LIN {X 0,Y 189.496,Z 286.196,A -85,B 0,C 180,E1 -22198.72,E2 -22198.72} C_VEL
LIN {X 0,Y 187.932,Z 288.132,A -85,B 0,C 180,E1 -22200.913,E2 -22200.913} C_VEL
LIN {X 0,Y 186.648,Z 289.597,A -85,B 0,C 180,E1 -22203.139,E2 -22203.139} C_VEL
LIN {X 0,Y 185.608,Z 290.594,A -85,B 0,C 180,E1 -22205.386,E2 -22205.386} C_VEL
LIN {X 0,Y 184.681,Z 291.189,A -85,B 0,C 180,E1 -22207.633,E2 -22207.633} C_VEL
LIN {X 0,Y 183.977,Z 291.376,A -85,B 0,C 180,E1 -22209.892,E2 -22209.892} C_VEL
LIN {X 0,Y 183.377,Z 290.818,A -85,B 0,C 180,E1 -22213.366,E2 -22213.366} C_VEL
LIN {X 0,Y 183.176,Z 289.357,A -85,B 0,C 180,E1 -22216.692,E2 -22216.692} C_VEL
LIN {X 0,Y 183.239,Z 287.851,A -85,B 0,C 180,E1 -22218.945,E2 -22218.945} C_VEL
LIN {X 0,Y 183.723,Z 284.759,A -85,B 0,C 180,E1 -22222.307,E2 -22222.307} C_VEL
LIN {X 0,Y 184.434,Z 280.616,A -85,B 0,C 180,E1 -22225.63,E2 -22225.63} C_VEL
LIN {X 0,Y 185.666,Z 274.289,A -85,B 0,C 180,E1 -22229.459,E2 -22229.459} C_VEL
LIN {X 0,Y 187.209,Z 267.409,A -85,B 0,C 180,E1 -22232.69,E2 -22232.69} C_VEL
LIN {X 0,Y 188.876,Z 260.381,A -85,B 0,C 180,E1 -22235.338,E2 -22235.338} C_VEL
LIN {X 0,Y 190.904,Z 251.904,A -85,B 0,C 180,E1 -22237.936,E2 -22237.936} C_VEL
LIN {X 0,Y 193.116,Z 241.454,A -85,B 0,C 180,E1 -22240.485,E2 -22240.485} C_VEL
LIN {X 0,Y 195.098,Z 231.113,A -85,B 0,C 180,E1 -22242.483,E2 -22242.483} C_VEL
LIN {X 0,Y 196.96,Z 219.8,A -85,B 0,C 180,E1 -22244.201,E2 -22244.201} C_VEL
LIN {X 0,Y 198.45,Z 208.263,A -85,B 0,C 180,E1 -22245.535,E2 -22245.535} C_VEL
LIN {X 0,Y 199.783,Z 194.686,A -85,B 0,C 180,E1 -22246.631,E2 -22246.631} C_VEL
LIN {X 0,Y 200.565,Z 181.404,A -85,B 0,C 180,E1 -22247.294,E2 -22247.294} C_VEL
LIN {X 0,Y 202.876,Z 125.441,A -85,B 0,C 180,E1 -22249.181,E2 -22249.181} C_VEL
LIN {X 0,Y 196.139,Z 109.947,A -85,B 0,C 180,E1 -22250.877,E2 -22250.877} C_VEL
LIN {X 0,Y 187.163,Z 92.933,A -85,B 0,C 180,E1 -22253.206,E2 -22253.206} C_VEL
LIN {X 0,Y 185.821,Z 90.28,A -85,B 0,C 180,E1 -22253.583,E2 -22253.583} C_VEL
LIN {X 0,Y 185.663,Z 89.355,A -85,B 0,C 180,E1 -22253.732,E2 -22253.732} C_VEL
LIN {X 0,Y 185.582,Z 89.366,A -85,B 0,C 180,E1 -22259.493,E2 -22259.493} C_VEL
LIN {X 0,Y 185.522,Z 89.36,A -85,B 0,C 180,E1 -22264.628,E2 -22264.628} C_VEL
LIN {X 0,Y 185.548,Z 89.372,A -85,B 0,C 180,E1 -22267.304,E2 -22267.304} C_VEL
LIN {X 0,Y 185.507,Z 89.372,A -85,B 0,C 180,E1 -22270.736,E2 -22270.736} C_VEL
LIN {X 0,Y 185.513,Z 89.371,A -85,B 0,C 180,E1 -22273.961,E2 -22273.961} C_VEL
LIN {X 0,Y 185.475,Z 89.376,A -85,B 0,C 180,E1 -22279.275,E2 -22279.275} C_VEL
LIN {X 0,Y 185.509,Z 89.34,A -85,B 0,C 180,E1 -22282.711,E2 -22282.711} C_VEL
LIN {X 0,Y 185.545,Z 89.356,A -85,B 0,C 180,E1 -22287.974,E2 -22287.974} C_VEL
LIN {X 0,Y 185.584,Z 89.366,A -85,B 0,C 180,E1 -22290.576,E2 -22290.576} C_VEL
LIN {X 0,Y 185.591,Z 89.352,A -85,B 0,C 180,E1 -22295.382,E2 -22295.382} C_VEL
LIN {X 0,Y 185.611,Z 89.365,A -85,B 0,C 180,E1 -22300.075,E2 -22300.075} C_VEL
LIN {X 0,Y 185.699,Z 89.342,A -85,B 0,C 180,E1 -22304.637,E2 -22304.637} C_VEL
LIN {X 0,Y 185.892,Z 89.327,A -85,B 0,C 180,E1 -22309.417,E2 -22309.417} C_VEL
LIN {X 0,Y 185.951,Z 89.313,A -85,B 0,C 180,E1 -22313.489,E2 -22313.489} C_VEL
LIN {X 0,Y 186.21,Z 89.286,A -85,B 0,C 180,E1 -22317.836,E2 -22317.836} C_VEL
LIN {X 0,Y 186.41,Z 89.252,A -85,B 0,C 180,E1 -22320,E2 -22320} C_VEL
LIN {X 0,Y 185.92,Z 89.325,A -85,B 0,C 180,E1 -22324.335,E2 -22324.335} C_VEL
LIN {X 0,Y 185.984,Z 89.307,A -85,B 0,C 180,E1 -22328.693,E2 -22328.693} C_VEL
LIN {X 0,Y 185.731,Z 89.348,A -85,B 0,C 180,E1 -22333.122,E2 -22333.122} C_VEL
LIN {X 0,Y 185.692,Z 89.353,A -85,B 0,C 180,E1 -22337.624,E2 -22337.624} C_VEL
LIN {X 0,Y 185.583,Z 89.365,A -85,B 0,C 180,E1 -22342.253,E2 -22342.253} C_VEL
LIN {X 0,Y 185.563,Z 89.37,A -85,B 0,C 180,E1 -22347.032,E2 -22347.032} C_VEL
LIN {X 0,Y 185.581,Z 89.358,A -85,B 0,C 180,E1 -22349.492,E2 -22349.492} C_VEL
LIN {X 0,Y 185.502,Z 89.377,A -85,B 0,C 180,E1 -22354.631,E2 -22354.631} C_VEL
LIN {X 0,Y 185.507,Z 89.377,A -85,B 0,C 180,E1 -22357.312,E2 -22357.312} C_VEL
LIN {X 0,Y 185.473,Z 89.38,A -85,B 0,C 180,E1 -22360.724,E2 -22360.724} C_VEL
LIN {X 0,Y 185.482,Z 89.373,A -85,B 0,C 180,E1 -22366.047,E2 -22366.047} C_VEL
LIN {X 0,Y 185.494,Z 89.51,A -85,B 0,C 180,E1 -22368.177,E2 -22368.177} C_VEL
LIN {X 0,Y 187.517,Z 97.408,A -85,B 0,C 180,E1 -22372.298,E2 -22372.298} C_VEL
LIN {X 0,Y 194.138,Z 113.363,A -85,B 0,C 180,E1 -22374.166,E2 -22374.166} C_VEL
LIN {X 0,Y 198.277,Z 124.653,A -85,B 0,C 180,E1 -22375.313,E2 -22375.313} C_VEL
LIN {X 0,Y 201.609,Z 160.671,A -85,B 0,C 180,E1 -22377.266,E2 -22377.266} C_VEL
LIN {X 0,Y 200.557,Z 187.322,A -85,B 0,C 180,E1 -22378.173,E2 -22378.173} C_VEL
LIN {X 0,Y 199.727,Z 193.163,A -85,B 0,C 180,E1 -22378.281,E2 -22378.281} C_VEL
LIN {X 0,Y 196.792,Z 202.635,A -85,B 0,C 180,E1 -22378.264,E2 -22378.264} C_VEL
LIN {X 0,Y 193.584,Z 212.011,A -85,B 0,C 180,E1 -22378.361,E2 -22378.361} C_VEL
LIN {X 0,Y 192.33,Z 217.701,A -85,B 0,C 180,E1 -22378.656,E2 -22378.656} C_VEL
LIN {X 0,Y 190.824,Z 229.613,A -85,B 0,C 180,E1 -22379.727,E2 -22379.727} C_VEL
LIN {X 0,Y 188.661,Z 242.542,A -85,B 0,C 180,E1 -22381.339,E2 -22381.339} C_VEL
LIN {X 0,Y 186.403,Z 253.251,A -85,B 0,C 180,E1 -22383.099,E2 -22383.099} C_VEL
LIN {X 0,Y 184.263,Z 263.146,A -85,B 0,C 180,E1 -22385.193,E2 -22385.193} C_VEL
LIN {X 0,Y 182.035,Z 272.867,A -85,B 0,C 180,E1 -22387.782,E2 -22387.782} C_VEL
LIN {X 0,Y 180.386,Z 279.889,A -85,B 0,C 180,E1 -22390.067,E2 -22390.067} C_VEL
LIN {X 0,Y 178.556,Z 288.207,A -85,B 0,C 180,E1 -22393.419,E2 -22393.419} C_VEL
LIN {X 0,Y 177.177,Z 294.878,A -85,B 0,C 180,E1 -22396.815,E2 -22396.815} C_VEL
LIN {X 0,Y 176.604,Z 299.374,A -85,B 0,C 180,E1 -22399.683,E2 -22399.683} C_VEL
LIN {X 0,Y 176.304,Z 303.668,A -85,B 0,C 180,E1 -22403.131,E2 -22403.131} C_VEL
LIN {X 0,Y 176.301,Z 305.931,A -85,B 0,C 180,E1 -22405.426,E2 -22405.426} C_VEL
LIN {X 0,Y 176.367,Z 307.699,A -85,B 0,C 180,E1 -22407.715,E2 -22407.715} C_VEL
LIN {X 0,Y 176.503,Z 309.022,A -85,B 0,C 180,E1 -22409.999,E2 -22409.999} C_VEL
LIN {X 0,Y 176.331,Z 309.912,A -85,B 0,C 180,E1 -22412.283,E2 -22412.283} C_VEL
LIN {X 0,Y 176.231,Z 310.408,A -85,B 0,C 180,E1 -22414.574,E2 -22414.574} C_VEL
LIN {X 0,Y 176.416,Z 310.152,A -85,B 0,C 180,E1 -22419.168,E2 -22419.168} C_VEL
LIN {X 0,Y 177.558,Z 308.367,A -85,B 0,C 180,E1 -22423.737,E2 -22423.737} C_VEL
LIN {X 0,Y 178.565,Z 306.883,A -85,B 0,C 180,E1 -22425.991,E2 -22425.991} C_VEL
LIN {X 0,Y 180.745,Z 303.862,A -85,B 0,C 180,E1 -22429.299,E2 -22429.299} C_VEL
LIN {X 0,Y 184.077,Z 298.833,A -85,B 0,C 180,E1 -22433.179,E2 -22433.179} C_VEL
LIN {X 0,Y 187.805,Z 292.664,A -85,B 0,C 180,E1 -22436.683,E2 -22436.683} C_VEL
LIN {X 0,Y 191.925,Z 285.778,A -85,B 0,C 180,E1 -22439.626,E2 -22439.626} C_VEL
LIN {X 0,Y 196.615,Z 277.218,A -85,B 0,C 180,E1 -22442.423,E2 -22442.423} C_VEL
LIN {X 0,Y 200.867,Z 268.468,A -85,B 0,C 180,E1 -22444.649,E2 -22444.649} C_VEL
LIN {X 0,Y 204.532,Z 260.069,A -85,B 0,C 180,E1 -22446.35,E2 -22446.35} C_VEL
LIN {X 0,Y 208.408,Z 249.896,A -85,B 0,C 180,E1 -22447.982,E2 -22447.982} C_VEL
LIN {X 0,Y 212.043,Z 238.795,A -85,B 0,C 180,E1 -22449.336,E2 -22449.336} C_VEL
LIN {X 0,Y 215.361,Z 226.423,A -85,B 0,C 180,E1 -22450.434,E2 -22450.434} C_VEL
LIN {X 0,Y 217.575,Z 214.056,A -85,B 0,C 180,E1 -22451.255,E2 -22451.255} C_VEL
LIN {X 0,Y 219.112,Z 200.89,A -85,B 0,C 180,E1 -22451.806,E2 -22451.806} C_VEL
LIN {X 0,Y 221.097,Z 169.395,A -85,B 0,C 180,E1 -22452.769,E2 -22452.769} C_VEL
LIN {X 0,Y 220.168,Z 161.646,A -85,B 0,C 180,E1 -22453.42,E2 -22453.42} C_VEL
LIN {X 0,Y 215.236,Z 149.691,A -85,B 0,C 180,E1 -22455.576,E2 -22455.576} C_VEL
LIN {X 0,Y 209.918,Z 138.652,A -85,B 0,C 180,E1 -22458.045,E2 -22458.045} C_VEL
LIN {X 0,Y 203.875,Z 127.771,A -85,B 0,C 180,E1 -22461.117,E2 -22461.117} C_VEL
LIN {X 0,Y 200.883,Z 122.753,A -85,B 0,C 180,E1 -22462.79,E2 -22462.79} C_VEL
LIN {X 0,Y 197.598,Z 117.462,A -85,B 0,C 180,E1 -22464.772,E2 -22464.772} C_VEL
LIN {X 0,Y 194.096,Z 112.066,A -85,B 0,C 180,E1 -22467.103,E2 -22467.103} C_VEL
LIN {X 0,Y 190.527,Z 106.917,A -85,B 0,C 180,E1 -22469.772,E2 -22469.772} C_VEL
LIN {X 0,Y 189.458,Z 105.438,A -85,B 0,C 180,E1 -22470.643,E2 -22470.643} C_VEL
LIN {X 0,Y 185.248,Z 99.511,A -85,B 0,C 180,E1 -22474.555,E2 -22474.555} C_VEL
LIN {X 0,Y 184.251,Z 98.309,A -85,B 0,C 180,E1 -22475.607,E2 -22475.607} C_VEL
LIN {X 0,Y 181.27,Z 94.972,A -85,B 0,C 180,E1 -22479.252,E2 -22479.252} C_VEL
LIN {X 0,Y 179.221,Z 92.29,A -85,B 0,C 180,E1 -22482.602,E2 -22482.602} C_VEL
LIN {X 0,Y 178.688,Z 90.572,A -85,B 0,C 180,E1 -22484.019,E2 -22484.019} C_VEL
LIN {X 0,Y 178.657,Z 90.226,A -85,B 0,C 180,E1 -22485.186,E2 -22485.186} C_VEL
LIN {X 0,Y 178.957,Z 90.181,A -85,B 0,C 180,E1 -22490.963,E2 -22490.963} C_VEL
LIN {X 0,Y 179.151,Z 90.15,A -85,B 0,C 180,E1 -22497.752,E2 -22497.752} C_VEL
LIN {X 0,Y 179.368,Z 90.141,A -85,B 0,C 180,E1 -22500.001,E2 -22500.001} C_VEL
LIN {X 0,Y 178.985,Z 90.178,A -85,B 0,C 180,E1 -22503.307,E2 -22503.307} C_VEL
LIN {X 0,Y 179.364,Z 92.055,A -85,B 0,C 180,E1 -22504.354,E2 -22504.354} C_VEL
LIN {X 0,Y 181.079,Z 94.465,A -85,B 0,C 180,E1 -22507.22,E2 -22507.22} C_VEL
LIN {X 0,Y 184.082,Z 96.395,A -85,B 0,C 180,E1 -22510.774,E2 -22510.774} C_VEL
LIN {X 0,Y 185.516,Z 99.384,A -85,B 0,C 180,E1 -22512.443,E2 -22512.443} C_VEL
LIN {X 0,Y 187.922,Z 101.543,A -85,B 0,C 180,E1 -22514.627,E2 -22514.627} C_VEL
LIN {X 0,Y 188.806,Z 102.204,A -85,B 0,C 180,E1 -22515.353,E2 -22515.353} C_VEL
LIN {X 0,Y 190.908,Z 105.519,A -85,B 0,C 180,E1 -22517.129,E2 -22517.129} C_VEL
LIN {X 0,Y 193.091,Z 107.65,A -85,B 0,C 180,E1 -22518.705,E2 -22518.705} C_VEL
LIN {X 0,Y 195.744,Z 111.352,A -85,B 0,C 180,E1 -22520.552,E2 -22520.552} C_VEL
LIN {X 0,Y 197.052,Z 112.765,A -85,B 0,C 180,E1 -22521.375,E2 -22521.375} C_VEL
LIN {X 0,Y 199.933,Z 116.546,A -85,B 0,C 180,E1 -22523.111,E2 -22523.111} C_VEL
LIN {X 0,Y 205.063,Z 123.799,A -85,B 0,C 180,E1 -22525.92,E2 -22525.92} C_VEL
LIN {X 0,Y 209.744,Z 130.716,A -85,B 0,C 180,E1 -22528.215,E2 -22528.215} C_VEL
LIN {X 0,Y 215.217,Z 139.457,A -85,B 0,C 180,E1 -22530.655,E2 -22530.655} C_VEL
LIN {X 0,Y 220.98,Z 149.875,A -85,B 0,C 180,E1 -22533.027,E2 -22533.027} C_VEL
LIN {X 0,Y 222.161,Z 152.174,A -85,B 0,C 180,E1 -22533.489,E2 -22533.489} C_VEL
LIN {X 0,Y 219.645,Z 189.927,A -85,B 0,C 180,E1 -22534.677,E2 -22534.677} C_VEL
LIN {X 0,Y 217.805,Z 203.659,A -85,B 0,C 180,E1 -22535.439,E2 -22535.439} C_VEL
LIN {X 0,Y 215.36,Z 216.368,A -85,B 0,C 180,E1 -22536.526,E2 -22536.526} C_VEL
LIN {X 0,Y 212.374,Z 227.641,A -85,B 0,C 180,E1 -22537.808,E2 -22537.808} C_VEL
LIN {X 0,Y 208.513,Z 239.481,A -85,B 0,C 180,E1 -22539.588,E2 -22539.588} C_VEL
LIN {X 0,Y 204.409,Z 249.786,A -85,B 0,C 180,E1 -22541.6,E2 -22541.6} C_VEL
LIN {X 0,Y 200.067,Z 259.097,A -85,B 0,C 180,E1 -22543.936,E2 -22543.936} C_VEL
LIN {X 0,Y 195.906,Z 266.984,A -85,B 0,C 180,E1 -22546.464,E2 -22546.464} C_VEL
LIN {X 0,Y 191.76,Z 274.127,A -85,B 0,C 180,E1 -22549.419,E2 -22549.419} C_VEL
LIN {X 0,Y 188.457,Z 279.189,A -85,B 0,C 180,E1 -22552.115,E2 -22552.115} C_VEL
LIN {X 0,Y 185.142,Z 283.802,A -85,B 0,C 180,E1 -22555.293,E2 -22555.293} C_VEL
LIN {X 0,Y 183.086,Z 286.374,A -85,B 0,C 180,E1 -22557.62,E2 -22557.62} C_VEL
LIN {X 0,Y 181.489,Z 288.257,A -85,B 0,C 180,E1 -22559.775,E2 -22559.775} C_VEL
LIN {X 0,Y 180.054,Z 289.805,A -85,B 0,C 180,E1 -22562.071,E2 -22562.071} C_VEL
LIN {X 0,Y 178.732,Z 290.986,A -85,B 0,C 180,E1 -22564.744,E2 -22564.744} C_VEL
LIN {X 0,Y 177.097,Z 291.753,A -85,B 0,C 180,E1 -22569.075,E2 -22569.075} C_VEL
LIN {X 0,Y 176.34,Z 291.203,A -85,B 0,C 180,E1 -22573.044,E2 -22573.044} C_VEL
LIN {X 0,Y 176.092,Z 289.919,A -85,B 0,C 180,E1 -22576.146,E2 -22576.146} C_VEL
LIN {X 0,Y 176.123,Z 288.494,A -85,B 0,C 180,E1 -22578.492,E2 -22578.492} C_VEL
LIN {X 0,Y 176.555,Z 285.497,A -85,B 0,C 180,E1 -22581.992,E2 -22581.992} C_VEL
LIN {X 0,Y 177.294,Z 281.461,A -85,B 0,C 180,E1 -22585.454,E2 -22585.454} C_VEL
LIN {X 0,Y 178.523,Z 275.271,A -85,B 0,C 180,E1 -22589.437,E2 -22589.437} C_VEL
LIN {X 0,Y 180.097,Z 268.52,A -85,B 0,C 180,E1 -22592.797,E2 -22592.797} C_VEL
LIN {X 0,Y 182.181,Z 260.138,A -85,B 0,C 180,E1 -22596.091,E2 -22596.091} C_VEL
LIN {X 0,Y 184.546,Z 250.418,A -85,B 0,C 180,E1 -22599.066,E2 -22599.066} C_VEL
LIN {X 0,Y 186.759,Z 240.313,A -85,B 0,C 180,E1 -22601.525,E2 -22601.525} C_VEL
LIN {X 0,Y 188.7,Z 230.329,A -85,B 0,C 180,E1 -22603.461,E2 -22603.461} C_VEL
LIN {X 0,Y 190.715,Z 218.615,A -85,B 0,C 180,E1 -22605.223,E2 -22605.223} C_VEL
LIN {X 0,Y 192.221,Z 206.531,A -85,B 0,C 180,E1 -22606.598,E2 -22606.598} C_VEL
LIN {X 0,Y 193.533,Z 193.209,A -85,B 0,C 180,E1 -22607.646,E2 -22607.646} C_VEL
LIN {X 0,Y 194.29,Z 179.563,A -85,B 0,C 180,E1 -22608.28,E2 -22608.28} C_VEL
LIN {X 0,Y 196.535,Z 127.249,A -85,B 0,C 180,E1 -22610.092,E2 -22610.092} C_VEL
LIN {X 0,Y 190.152,Z 112.596,A -85,B 0,C 180,E1 -22611.791,E2 -22611.791} C_VEL
LIN {X 0,Y 181.659,Z 96.589,A -85,B 0,C 180,E1 -22614.117,E2 -22614.117} C_VEL
LIN {X 0,Y 180.081,Z 93.814,A -85,B 0,C 180,E1 -22614.57,E2 -22614.57} C_VEL
LIN {X 0,Y 178.751,Z 91.288,A -85,B 0,C 180,E1 -22614.97,E2 -22614.97} C_VEL
LIN {X 0,Y 178.524,Z 90.248,A -85,B 0,C 180,E1 -22615.115,E2 -22615.115} C_VEL
LIN {X 0,Y 178.526,Z 90.248,A -85,B 0,C 180,E1 -22619.993,E2 -22619.993} C_VEL
LIN {X 0,Y 178.499,Z 90.232,A -85,B 0,C 180,E1 -22624.224,E2 -22624.224} C_VEL
LIN {X 0,Y 178.43,Z 90.255,A -85,B 0,C 180,E1 -22629.066,E2 -22629.066} C_VEL
LIN {X 0,Y 178.434,Z 90.258,A -85,B 0,C 180,E1 -22632.036,E2 -22632.036} C_VEL
LIN {X 0,Y 178.426,Z 90.25,A -85,B 0,C 180,E1 -22635.155,E2 -22635.155} C_VEL
LIN {X 0,Y 178.413,Z 90.258,A -85,B 0,C 180,E1 -22638.457,E2 -22638.457} C_VEL
LIN {X 0,Y 178.425,Z 90.212,A -85,B 0,C 180,E1 -22643.783,E2 -22643.783} C_VEL
LIN {X 0,Y 178.489,Z 90.217,A -85,B 0,C 180,E1 -22646.546,E2 -22646.546} C_VEL
LIN {X 0,Y 178.525,Z 90.243,A -85,B 0,C 180,E1 -22650.007,E2 -22650.007} C_VEL
LIN {X 0,Y 178.538,Z 90.232,A -85,B 0,C 180,E1 -22654.875,E2 -22654.875} C_VEL
LIN {X 0,Y 178.627,Z 90.232,A -85,B 0,C 180,E1 -22660.783,E2 -22660.783} C_VEL
LIN {X 0,Y 178.662,Z 90.226,A -85,B 0,C 180,E1 -22666.348,E2 -22666.348} C_VEL
LIN {X 0,Y 178.915,Z 90.188,A -85,B 0,C 180,E1 -22670.959,E2 -22670.959} C_VEL
LIN {X 0,Y 179.155,Z 90.165,A -85,B 0,C 180,E1 -22677.751,E2 -22677.751} C_VEL
LIN {X 0,Y 179.373,Z 90.128,A -85,B 0,C 180,E1 -22679.999,E2 -22679.999} C_VEL
LIN {X 0,Y 178.868,Z 90.203,A -85,B 0,C 180,E1 -22684.507,E2 -22684.507} C_VEL
LIN {X 0,Y 178.913,Z 90.188,A -85,B 0,C 180,E1 -22689.04,E2 -22689.04} C_VEL
LIN {X 0,Y 178.659,Z 90.226,A -85,B 0,C 180,E1 -22693.652,E2 -22693.652} C_VEL
LIN {X 0,Y 178.625,Z 90.236,A -85,B 0,C 180,E1 -22699.215,E2 -22699.215} C_VEL
LIN {X 0,Y 178.522,Z 90.243,A -85,B 0,C 180,E1 -22705.114,E2 -22705.114} C_VEL
LIN {X 0,Y 178.525,Z 90.235,A -85,B 0,C 180,E1 -22709.993,E2 -22709.993} C_VEL
LIN {X 0,Y 178.487,Z 90.251,A -85,B 0,C 180,E1 -22714.219,E2 -22714.219} C_VEL
LIN {X 0,Y 178.397,Z 90.261,A -85,B 0,C 180,E1 -22719.074,E2 -22719.074} C_VEL
LIN {X 0,Y 178.4,Z 90.263,A -85,B 0,C 180,E1 -22722.044,E2 -22722.044} C_VEL
LIN {X 0,Y 178.451,Z 90.407,A -85,B 0,C 180,E1 -22727.215,E2 -22727.215} C_VEL
LIN {X 0,Y 180.207,Z 97.099,A -85,B 0,C 180,E1 -22730.848,E2 -22730.848} C_VEL
LIN {X 0,Y 186.959,Z 112.594,A -85,B 0,C 180,E1 -22732.871,E2 -22732.871} C_VEL
LIN {X 0,Y 192.111,Z 126.464,A -85,B 0,C 180,E1 -22734.381,E2 -22734.381} C_VEL
LIN {X 0,Y 195.261,Z 160.573,A -85,B 0,C 180,E1 -22736.32,E2 -22736.32} C_VEL
LIN {X 0,Y 193.234,Z 207.375,A -85,B 0,C 180,E1 -22738.018,E2 -22738.018} C_VEL
LIN {X 0,Y 192.33,Z 217.701,A -85,B 0,C 180,E1 -22738.656,E2 -22738.656} C_VEL
LIN {X 0,Y 191.474,Z 221.466,A -85,B 0,C 180,E1 -22738.896,E2 -22738.896} C_VEL
LIN {X 0,Y 188.656,Z 228.732,A -85,B 0,C 180,E1 -22739.327,E2 -22739.327} C_VEL
LIN {X 0,Y 183.643,Z 239.211,A -85,B 0,C 180,E1 -22740.161,E2 -22740.161} C_VEL
LIN {X 0,Y 181.743,Z 244.423,A -85,B 0,C 180,E1 -22740.82,E2 -22740.82} C_VEL
LIN {X 0,Y 181.308,Z 246.12,A -85,B 0,C 180,E1 -22741.086,E2 -22741.086} C_VEL
LIN {X 0,Y 178.97,Z 257.103,A -85,B 0,C 180,E1 -22743.153,E2 -22743.153} C_VEL
LIN {X 0,Y 176.808,Z 266.257,A -85,B 0,C 180,E1 -22745.331,E2 -22745.331} C_VEL
LIN {X 0,Y 174.491,Z 275.177,A -85,B 0,C 180,E1 -22747.961,E2 -22747.961} C_VEL
LIN {X 0,Y 172.581,Z 283.343,A -85,B 0,C 180,E1 -22750.986,E2 -22750.986} C_VEL
LIN {X 0,Y 170.895,Z 290.898,A -85,B 0,C 180,E1 -22754.495,E2 -22754.495} C_VEL
LIN {X 0,Y 169.782,Z 296.95,A -85,B 0,C 180,E1 -22758.054,E2 -22758.054} C_VEL
LIN {X 0,Y 169.287,Z 301.72,A -85,B 0,C 180,E1 -22761.644,E2 -22761.644} C_VEL
LIN {X 0,Y 169.256,Z 305.339,A -85,B 0,C 180,E1 -22765.235,E2 -22765.235} C_VEL
LIN {X 0,Y 169.284,Z 307.171,A -85,B 0,C 180,E1 -22767.62,E2 -22767.62} C_VEL
LIN {X 0,Y 169.436,Z 308.528,A -85,B 0,C 180,E1 -22769.999,E2 -22769.999} C_VEL
LIN {X 0,Y 169.153,Z 309.899,A -85,B 0,C 180,E1 -22774.327,E2 -22774.327} C_VEL
LIN {X 0,Y 169.111,Z 310.102,A -85,B 0,C 180,E1 -22777.161,E2 -22777.161} C_VEL
LIN {X 0,Y 169.888,Z 309.14,A -85,B 0,C 180,E1 -22781.936,E2 -22781.936} C_VEL
LIN {X 0,Y 171.737,Z 306.658,A -85,B 0,C 180,E1 -22786.645,E2 -22786.645} C_VEL
LIN {X 0,Y 174.015,Z 303.693,A -85,B 0,C 180,E1 -22790.077,E2 -22790.077} C_VEL
LIN {X 0,Y 176.9,Z 299.726,A -85,B 0,C 180,E1 -22793.408,E2 -22793.408} C_VEL
LIN {X 0,Y 180.216,Z 294.661,A -85,B 0,C 180,E1 -22796.645,E2 -22796.645} C_VEL
LIN {X 0,Y 184.271,Z 288.346,A -85,B 0,C 180,E1 -22799.722,E2 -22799.722} C_VEL
LIN {X 0,Y 188.966,Z 280.483,A -85,B 0,C 180,E1 -22802.634,E2 -22802.634} C_VEL
LIN {X 0,Y 194.096,Z 270.728,A -85,B 0,C 180,E1 -22805.403,E2 -22805.403} C_VEL
LIN {X 0,Y 198.886,Z 260.633,A -85,B 0,C 180,E1 -22807.557,E2 -22807.557} C_VEL
LIN {X 0,Y 203.43,Z 249.24,A -85,B 0,C 180,E1 -22809.405,E2 -22809.405} C_VEL
LIN {X 0,Y 207.19,Z 238.076,A -85,B 0,C 180,E1 -22810.765,E2 -22810.765} C_VEL
LIN {X 0,Y 210.56,Z 225.576,A -85,B 0,C 180,E1 -22811.877,E2 -22811.877} C_VEL
LIN {X 0,Y 213.015,Z 212.226,A -85,B 0,C 180,E1 -22812.729,E2 -22812.729} C_VEL
LIN {X 0,Y 214.469,Z 199.358,A -85,B 0,C 180,E1 -22813.25,E2 -22813.25} C_VEL
LIN {X 0,Y 216.359,Z 170.637,A -85,B 0,C 180,E1 -22814.127,E2 -22814.127} C_VEL
LIN {X 0,Y 215.671,Z 164.769,A -85,B 0,C 180,E1 -22814.646,E2 -22814.646} C_VEL
LIN {X 0,Y 210.864,Z 152.977,A -85,B 0,C 180,E1 -22816.894,E2 -22816.894} C_VEL
LIN {X 0,Y 206.363,Z 143.506,A -85,B 0,C 180,E1 -22819.117,E2 -22819.117} C_VEL
LIN {X 0,Y 200.898,Z 133.302,A -85,B 0,C 180,E1 -22822.072,E2 -22822.072} C_VEL
LIN {X 0,Y 198.165,Z 128.524,A -85,B 0,C 180,E1 -22823.69,E2 -22823.69} C_VEL
LIN {X 0,Y 195.199,Z 123.575,A -85,B 0,C 180,E1 -22825.576,E2 -22825.576} C_VEL
LIN {X 0,Y 191.685,Z 118,A -85,B 0,C 180,E1 -22828.059,E2 -22828.059} C_VEL
LIN {X 0,Y 188.201,Z 112.612,A -85,B 0,C 180,E1 -22830.852,E2 -22830.852} C_VEL
LIN {X 0,Y 183.558,Z 105.969,A -85,B 0,C 180,E1 -22835.319,E2 -22835.319} C_VEL
LIN {X 0,Y 180.055,Z 101.846,A -85,B 0,C 180,E1 -22839.66,E2 -22839.66} C_VEL
LIN {X 0,Y 177.951,Z 98.869,A -85,B 0,C 180,E1 -22843.362,E2 -22843.362} C_VEL
LIN {X 0,Y 177.417,Z 97.247,A -85,B 0,C 180,E1 -22844.786,E2 -22844.786} C_VEL
LIN {X 0,Y 175.465,Z 96.384,A -85,B 0,C 180,E1 -22853.099,E2 -22853.099} C_VEL
LIN {X 0,Y 177.072,Z 96.912,A -85,B 0,C 180,E1 -22861.138,E2 -22861.138} C_VEL
LIN {X 0,Y 177.763,Z 97.286,A -85,B 0,C 180,E1 -22862.691,E2 -22862.691} C_VEL
LIN {X 0,Y 178.516,Z 99.58,A -85,B 0,C 180,E1 -22864.517,E2 -22864.517} C_VEL
LIN {X 0,Y 180.822,Z 102.098,A -85,B 0,C 180,E1 -22868.1,E2 -22868.1} C_VEL
LIN {X 0,Y 182.531,Z 103.253,A -85,B 0,C 180,E1 -22870.126,E2 -22870.126} C_VEL
LIN {X 0,Y 184.241,Z 106.391,A -85,B 0,C 180,E1 -22872.129,E2 -22872.129} C_VEL
LIN {X 0,Y 187.041,Z 108.909,A -85,B 0,C 180,E1 -22874.702,E2 -22874.702} C_VEL
LIN {X 0,Y 189.513,Z 112.52,A -85,B 0,C 180,E1 -22876.828,E2 -22876.828} C_VEL
LIN {X 0,Y 191.163,Z 114.294,A -85,B 0,C 180,E1 -22878.072,E2 -22878.072} C_VEL
LIN {X 0,Y 193.984,Z 118.05,A -85,B 0,C 180,E1 -22880.089,E2 -22880.089} C_VEL
LIN {X 0,Y 198.456,Z 124.157,A -85,B 0,C 180,E1 -22882.927,E2 -22882.927} C_VEL
LIN {X 0,Y 202.332,Z 129.685,A -85,B 0,C 180,E1 -22885.115,E2 -22885.115} C_VEL
LIN {X 0,Y 207.264,Z 137.224,A -85,B 0,C 180,E1 -22887.645,E2 -22887.645} C_VEL
LIN {X 0,Y 212.742,Z 146.379,A -85,B 0,C 180,E1 -22890.183,E2 -22890.183} C_VEL
LIN {X 0,Y 217.378,Z 155.111,A -85,B 0,C 180,E1 -22892.18,E2 -22892.18} C_VEL
LIN {X 0,Y 214.885,Z 190.321,A -85,B 0,C 180,E1 -22893.291,E2 -22893.291} C_VEL
LIN {X 0,Y 213,Z 203.916,A -85,B 0,C 180,E1 -22894.05,E2 -22894.05} C_VEL
LIN {X 0,Y 210.515,Z 216.444,A -85,B 0,C 180,E1 -22895.123,E2 -22895.123} C_VEL
LIN {X 0,Y 207.414,Z 227.78,A -85,B 0,C 180,E1 -22896.416,E2 -22896.416} C_VEL
LIN {X 0,Y 203.751,Z 238.706,A -85,B 0,C 180,E1 -22898.052,E2 -22898.052} C_VEL
LIN {X 0,Y 199.571,Z 248.975,A -85,B 0,C 180,E1 -22900.011,E2 -22900.011} C_VEL
LIN {X 0,Y 195.013,Z 258.517,A -85,B 0,C 180,E1 -22902.373,E2 -22902.373} C_VEL
LIN {X 0,Y 190.993,Z 265.923,A -85,B 0,C 180,E1 -22904.7,E2 -22904.7} C_VEL
LIN {X 0,Y 186.87,Z 272.709,A -85,B 0,C 180,E1 -22907.394,E2 -22907.394} C_VEL
LIN {X 0,Y 182.437,Z 279.33,A -85,B 0,C 180,E1 -22910.85,E2 -22910.85} C_VEL
LIN {X 0,Y 179.087,Z 283.772,A -85,B 0,C 180,E1 -22913.94,E2 -22913.94} C_VEL
LIN {X 0,Y 176.565,Z 286.8,A -85,B 0,C 180,E1 -22916.709,E2 -22916.709} C_VEL
LIN {X 0,Y 173.526,Z 289.987,A -85,B 0,C 180,E1 -22920.922,E2 -22920.922} C_VEL
LIN {X 0,Y 171.844,Z 291.404,A -85,B 0,C 180,E1 -22924.126,E2 -22924.126} C_VEL
LIN {X 0,Y 170.24,Z 292.126,A -85,B 0,C 180,E1 -22928.19,E2 -22928.19} C_VEL
LIN {X 0,Y 169.288,Z 291.582,A -85,B 0,C 180,E1 -22932.719,E2 -22932.719} C_VEL
LIN {X 0,Y 169.031,Z 290.481,A -85,B 0,C 180,E1 -22935.555,E2 -22935.555} C_VEL
LIN {X 0,Y 168.998,Z 289.106,A -85,B 0,C 180,E1 -22938,E2 -22938} C_VEL
LIN {X 0,Y 169.399,Z 286.205,A -85,B 0,C 180,E1 -22941.652,E2 -22941.652} C_VEL
LIN {X 0,Y 170.153,Z 282.27,A -85,B 0,C 180,E1 -22945.262,E2 -22945.262} C_VEL
LIN {X 0,Y 171.198,Z 277.212,A -85,B 0,C 180,E1 -22948.825,E2 -22948.825} C_VEL
LIN {X 0,Y 172.668,Z 270.866,A -85,B 0,C 180,E1 -22952.334,E2 -22952.334} C_VEL
LIN {X 0,Y 174.689,Z 262.905,A -85,B 0,C 180,E1 -22955.773,E2 -22955.773} C_VEL
LIN {X 0,Y 176.798,Z 254.784,A -85,B 0,C 180,E1 -22958.574,E2 -22958.574} C_VEL
LIN {X 0,Y 179.202,Z 244.889,A -85,B 0,C 180,E1 -22961.309,E2 -22961.309} C_VEL
LIN {X 0,Y 181.574,Z 233.794,A -85,B 0,C 180,E1 -22963.715,E2 -22963.715} C_VEL
LIN {X 0,Y 183.528,Z 222.949,A -85,B 0,C 180,E1 -22965.549,E2 -22965.549} C_VEL
LIN {X 0,Y 185.345,Z 210.984,A -85,B 0,C 180,E1 -22967.09,E2 -22967.09} C_VEL
LIN {X 0,Y 186.798,Z 198.494,A -85,B 0,C 180,E1 -22968.249,E2 -22968.249} C_VEL
LIN {X 0,Y 187.704,Z 185.85,A -85,B 0,C 180,E1 -22969.01,E2 -22969.01} C_VEL
LIN {X 0,Y 190.333,Z 129.182,A -85,B 0,C 180,E1 -22971.041,E2 -22971.041} C_VEL
LIN {X 0,Y 184.337,Z 115.468,A -85,B 0,C 180,E1 -22972.727,E2 -22972.727} C_VEL
LIN {X 0,Y 175.556,Z 98.831,A -85,B 0,C 180,E1 -22975.294,E2 -22975.294} C_VEL
LIN {X 0,Y 172.903,Z 94.619,A -85,B 0,C 180,E1 -22976.096,E2 -22976.096} C_VEL
LIN {X 0,Y 171.678,Z 92.283,A -85,B 0,C 180,E1 -22976.498,E2 -22976.498} C_VEL
LIN {X 0,Y 171.417,Z 91.12,A -85,B 0,C 180,E1 -22976.63,E2 -22976.63} C_VEL
LIN {X 0,Y 171.444,Z 91.129,A -85,B 0,C 180,E1 -22980.586,E2 -22980.586} C_VEL
LIN {X 0,Y 171.41,Z 91.119,A -85,B 0,C 180,E1 -22985.032,E2 -22985.032} C_VEL
LIN {X 0,Y 171.39,Z 91.134,A -85,B 0,C 180,E1 -22988.819,E2 -22988.819} C_VEL
LIN {X 0,Y 171.352,Z 91.134,A -85,B 0,C 180,E1 -22994.208,E2 -22994.208} C_VEL
LIN {X 0,Y 171.343,Z 91.138,A -85,B 0,C 180,E1 -22998.983,E2 -22998.983} C_VEL
LIN {X 0,Y 171.39,Z 91.102,A -85,B 0,C 180,E1 -23002.041,E2 -23002.041} C_VEL
LIN {X 0,Y 171.401,Z 91.085,A -85,B 0,C 180,E1 -23005.092,E2 -23005.092} C_VEL
LIN {X 0,Y 171.452,Z 91.126,A -85,B 0,C 180,E1 -23010.534,E2 -23010.534} C_VEL
LIN {X 0,Y 171.461,Z 91.111,A -85,B 0,C 180,E1 -23015.801,E2 -23015.801} C_VEL
LIN {X 0,Y 171.583,Z 91.109,A -85,B 0,C 180,E1 -23020.871,E2 -23020.871} C_VEL
LIN {X 0,Y 171.58,Z 91.105,A -85,B 0,C 180,E1 -23025.772,E2 -23025.772} C_VEL
LIN {X 0,Y 171.851,Z 91.068,A -85,B 0,C 180,E1 -23030.584,E2 -23030.584} C_VEL
LIN {X 0,Y 171.819,Z 91.08,A -85,B 0,C 180,E1 -23035.307,E2 -23035.307} C_VEL
LIN {X 0,Y 172.336,Z 91.004,A -85,B 0,C 180,E1 -23039.999,E2 -23039.999} C_VEL
LIN {X 0,Y 171.816,Z 91.082,A -85,B 0,C 180,E1 -23044.692,E2 -23044.692} C_VEL
LIN {X 0,Y 171.85,Z 91.069,A -85,B 0,C 180,E1 -23049.415,E2 -23049.415} C_VEL
LIN {X 0,Y 171.578,Z 91.107,A -85,B 0,C 180,E1 -23054.227,E2 -23054.227} C_VEL
LIN {X 0,Y 171.544,Z 91.116,A -85,B 0,C 180,E1 -23059.559,E2 -23059.559} C_VEL
LIN {X 0,Y 171.461,Z 91.123,A -85,B 0,C 180,E1 -23065.609,E2 -23065.609} C_VEL
LIN {X 0,Y 171.444,Z 91.116,A -85,B 0,C 180,E1 -23070.586,E2 -23070.586} C_VEL
LIN {X 0,Y 171.395,Z 91.134,A -85,B 0,C 180,E1 -23075.034,E2 -23075.034} C_VEL
LIN {X 0,Y 171.359,Z 91.138,A -85,B 0,C 180,E1 -23078.807,E2 -23078.807} C_VEL
LIN {X 0,Y 171.326,Z 91.128,A -85,B 0,C 180,E1 -23084.215,E2 -23084.215} C_VEL
LIN {X 0,Y 171.374,Z 91.174,A -85,B 0,C 180,E1 -23086.085,E2 -23086.085} C_VEL
LIN {X 0,Y 172.714,Z 96.457,A -85,B 0,C 180,E1 -23089.185,E2 -23089.185} C_VEL
LIN {X 0,Y 178.847,Z 109.759,A -85,B 0,C 180,E1 -23091.166,E2 -23091.166} C_VEL
LIN {X 0,Y 185.082,Z 125.765,A -85,B 0,C 180,E1 -23093.114,E2 -23093.114} C_VEL
LIN {X 0,Y 186.218,Z 129.898,A -85,B 0,C 180,E1 -23093.505,E2 -23093.505} C_VEL
LIN {X 0,Y 188.993,Z 161.426,A -85,B 0,C 180,E1 -23095.356,E2 -23095.356} C_VEL
LIN {X 0,Y 186.963,Z 206.218,A -85,B 0,C 180,E1 -23097.009,E2 -23097.009} C_VEL
LIN {X 0,Y 185.624,Z 219.905,A -85,B 0,C 180,E1 -23097.912,E2 -23097.912} C_VEL
LIN {X 0,Y 183.974,Z 231.991,A -85,B 0,C 180,E1 -23099.113,E2 -23099.113} C_VEL
LIN {X 0,Y 181.748,Z 244.186,A -85,B 0,C 180,E1 -23100.777,E2 -23100.777} C_VEL
LIN {X 0,Y 181.308,Z 246.12,A -85,B 0,C 180,E1 -23101.086,E2 -23101.086} C_VEL
LIN {X 0,Y 179.603,Z 251.191,A -85,B 0,C 180,E1 -23101.886,E2 -23101.886} C_VEL
LIN {X 0,Y 175.173,Z 259.09,A -85,B 0,C 180,E1 -23103.192,E2 -23103.192} C_VEL
LIN {X 0,Y 170.666,Z 266.504,A -85,B 0,C 180,E1 -23104.777,E2 -23104.777} C_VEL
LIN {X 0,Y 168.874,Z 270.813,A -85,B 0,C 180,E1 -23105.999,E2 -23105.999} C_VEL
LIN {X 0,Y 166.873,Z 277.87,A -85,B 0,C 180,E1 -23108.375,E2 -23108.375} C_VEL
LIN {X 0,Y 165.15,Z 285.163,A -85,B 0,C 180,E1 -23111.387,E2 -23111.387} C_VEL
LIN {X 0,Y 163.512,Z 292.277,A -85,B 0,C 180,E1 -23115.054,E2 -23115.054} C_VEL
LIN {X 0,Y 162.551,Z 297.957,A -85,B 0,C 180,E1 -23118.78,E2 -23118.78} C_VEL
LIN {X 0,Y 162.158,Z 302.404,A -85,B 0,C 180,E1 -23122.528,E2 -23122.528} C_VEL
LIN {X 0,Y 162.161,Z 305.082,A -85,B 0,C 180,E1 -23125.422,E2 -23125.422} C_VEL
LIN {X 0,Y 162.205,Z 306.626,A -85,B 0,C 180,E1 -23127.516,E2 -23127.516} C_VEL
LIN {X 0,Y 162.37,Z 308.033,A -85,B 0,C 180,E1 -23129.999,E2 -23129.999} C_VEL
LIN {X 0,Y 162.082,Z 309.416,A -85,B 0,C 180,E1 -23134.214,E2 -23134.214} C_VEL
LIN {X 0,Y 162.037,Z 309.707,A -85,B 0,C 180,E1 -23137.476,E2 -23137.476} C_VEL
LIN {X 0,Y 162.35,Z 309.473,A -85,B 0,C 180,E1 -23139.97,E2 -23139.97} C_VEL
LIN {X 0,Y 163.712,Z 307.816,A -85,B 0,C 180,E1 -23144.925,E2 -23144.925} C_VEL
LIN {X 0,Y 164.938,Z 306.42,A -85,B 0,C 180,E1 -23147.353,E2 -23147.353} C_VEL
LIN {X 0,Y 167.325,Z 303.522,A -85,B 0,C 180,E1 -23150.916,E2 -23150.916} C_VEL
LIN {X 0,Y 170.369,Z 299.629,A -85,B 0,C 180,E1 -23154.362,E2 -23154.362} C_VEL
LIN {X 0,Y 173.884,Z 294.641,A -85,B 0,C 180,E1 -23157.697,E2 -23157.697} C_VEL
LIN {X 0,Y 178.129,Z 288.414,A -85,B 0,C 180,E1 -23160.857,E2 -23160.857} C_VEL
LIN {X 0,Y 183.038,Z 280.698,A -85,B 0,C 180,E1 -23163.83,E2 -23163.83} C_VEL
LIN {X 0,Y 188.361,Z 271.064,A -85,B 0,C 180,E1 -23166.653,E2 -23166.653} C_VEL
LIN {X 0,Y 193.312,Z 261.154,A -85,B 0,C 180,E1 -23168.838,E2 -23168.838} C_VEL
LIN {X 0,Y 198.02,Z 250.024,A -85,B 0,C 180,E1 -23170.703,E2 -23170.703} C_VEL
LIN {X 0,Y 201.901,Z 239.144,A -85,B 0,C 180,E1 -23172.072,E2 -23172.072} C_VEL
LIN {X 0,Y 205.399,Z 227.132,A -85,B 0,C 180,E1 -23173.182,E2 -23173.182} C_VEL
LIN {X 0,Y 207.943,Z 214.632,A -85,B 0,C 180,E1 -23174.054,E2 -23174.054} C_VEL
LIN {X 0,Y 209.624,Z 202.162,A -85,B 0,C 180,E1 -23174.606,E2 -23174.606} C_VEL
LIN {X 0,Y 211.741,Z 171.94,A -85,B 0,C 180,E1 -23175.555,E2 -23175.555} C_VEL
LIN {X 0,Y 211.336,Z 168.066,A -85,B 0,C 180,E1 -23175.901,E2 -23175.901} C_VEL
LIN {X 0,Y 206.337,Z 155.609,A -85,B 0,C 180,E1 -23178.408,E2 -23178.408} C_VEL
LIN {X 0,Y 202.042,Z 146.653,A -85,B 0,C 180,E1 -23180.695,E2 -23180.695} C_VEL
LIN {X 0,Y 197.699,Z 138.28,A -85,B 0,C 180,E1 -23183.228,E2 -23183.228} C_VEL
LIN {X 0,Y 194.953,Z 133.398,A -85,B 0,C 180,E1 -23184.964,E2 -23184.964} C_VEL
LIN {X 0,Y 192.34,Z 128.863,A -85,B 0,C 180,E1 -23186.764,E2 -23186.764} C_VEL
LIN {X 0,Y 189.491,Z 124.154,A -85,B 0,C 180,E1 -23188.91,E2 -23188.91} C_VEL
LIN {X 0,Y 185.604,Z 118.097,A -85,B 0,C 180,E1 -23192.24,E2 -23192.24} C_VEL
LIN {X 0,Y 181.474,Z 111.883,A -85,B 0,C 180,E1 -23196.594,E2 -23196.594} C_VEL
LIN {X 0,Y 178.774,Z 108.668,A -85,B 0,C 180,E1 -23200.19,E2 -23200.19} C_VEL
LIN {X 0,Y 176.783,Z 105.632,A -85,B 0,C 180,E1 -23203.954,E2 -23203.954} C_VEL
LIN {X 0,Y 176.257,Z 104.191,A -85,B 0,C 180,E1 -23205.422,E2 -23205.422} C_VEL
LIN {X 0,Y 174.592,Z 103.407,A -85,B 0,C 180,E1 -23213.064,E2 -23213.064} C_VEL
LIN {X 0,Y 176.567,Z 104.069,A -85,B 0,C 180,E1 -23221.996,E2 -23221.996} C_VEL
LIN {X 0,Y 177.522,Z 106.723,A -85,B 0,C 180,E1 -23224.364,E2 -23224.364} C_VEL
LIN {X 0,Y 180.042,Z 109.294,A -85,B 0,C 180,E1 -23228.277,E2 -23228.277} C_VEL
LIN {X 0,Y 181.045,Z 110.058,A -85,B 0,C 180,E1 -23229.501,E2 -23229.501} C_VEL
LIN {X 0,Y 182.971,Z 113.39,A -85,B 0,C 180,E1 -23231.81,E2 -23231.81} C_VEL
LIN {X 0,Y 185.333,Z 115.625,A -85,B 0,C 180,E1 -23234.069,E2 -23234.069} C_VEL
LIN {X 0,Y 187.997,Z 119.37,A -85,B 0,C 180,E1 -23236.427,E2 -23236.427} C_VEL
LIN {X 0,Y 189.167,Z 120.756,A -85,B 0,C 180,E1 -23237.352,E2 -23237.352} C_VEL
LIN {X 0,Y 192.191,Z 124.724,A -85,B 0,C 180,E1 -23239.589,E2 -23239.589} C_VEL
LIN {X 0,Y 196.455,Z 130.941,A -85,B 0,C 180,E1 -23242.415,E2 -23242.415} C_VEL
LIN {X 0,Y 201.101,Z 137.756,A -85,B 0,C 180,E1 -23245.098,E2 -23245.098} C_VEL
LIN {X 0,Y 207.122,Z 147.645,A -85,B 0,C 180,E1 -23248.208,E2 -23248.208} C_VEL
LIN {X 0,Y 212.682,Z 157.909,A -85,B 0,C 180,E1 -23250.789,E2 -23250.789} C_VEL
LIN {X 0,Y 210.286,Z 190.642,A -85,B 0,C 180,E1 -23251.839,E2 -23251.839} C_VEL
LIN {X 0,Y 208.269,Z 204.62,A -85,B 0,C 180,E1 -23252.626,E2 -23252.626} C_VEL
LIN {X 0,Y 205.581,Z 217.399,A -85,B 0,C 180,E1 -23253.741,E2 -23253.741} C_VEL
LIN {X 0,Y 202.054,Z 229.599,A -85,B 0,C 180,E1 -23255.177,E2 -23255.177} C_VEL
LIN {X 0,Y 198.261,Z 240.202,A -85,B 0,C 180,E1 -23256.817,E2 -23256.817} C_VEL
LIN {X 0,Y 193.91,Z 250.265,A -85,B 0,C 180,E1 -23258.811,E2 -23258.811} C_VEL
LIN {X 0,Y 189.174,Z 259.62,A -85,B 0,C 180,E1 -23261.211,E2 -23261.211} C_VEL
LIN {X 0,Y 184.767,Z 267.274,A -85,B 0,C 180,E1 -23263.723,E2 -23263.723} C_VEL
LIN {X 0,Y 179.958,Z 274.728,A -85,B 0,C 180,E1 -23266.888,E2 -23266.888} C_VEL
LIN {X 0,Y 175.699,Z 280.596,A -85,B 0,C 180,E1 -23270.209,E2 -23270.209} C_VEL
LIN {X 0,Y 171.959,Z 285.137,A -85,B 0,C 180,E1 -23273.658,E2 -23273.658} C_VEL
LIN {X 0,Y 168.841,Z 288.519,A -85,B 0,C 180,E1 -23277.241,E2 -23277.241} C_VEL
LIN {X 0,Y 167.097,Z 290.168,A -85,B 0,C 180,E1 -23279.689,E2 -23279.689} C_VEL
LIN {X 0,Y 165.012,Z 291.814,A -85,B 0,C 180,E1 -23283.434,E2 -23283.434} C_VEL
LIN {X 0,Y 163.422,Z 292.499,A -85,B 0,C 180,E1 -23287.23,E2 -23287.23} C_VEL
LIN {X 0,Y 162.712,Z 292.432,A -85,B 0,C 180,E1 -23289.786,E2 -23289.786} C_VEL
LIN {X 0,Y 162.256,Z 291.963,A -85,B 0,C 180,E1 -23292.351,E2 -23292.351} C_VEL
LIN {X 0,Y 161.96,Z 291.042,A -85,B 0,C 180,E1 -23294.91,E2 -23294.91} C_VEL
LIN {X 0,Y 161.886,Z 289.713,A -85,B 0,C 180,E1 -23297.464,E2 -23297.464} C_VEL
LIN {X 0,Y 162.233,Z 286.908,A -85,B 0,C 180,E1 -23301.28,E2 -23301.28} C_VEL
LIN {X 0,Y 162.978,Z 283.074,A -85,B 0,C 180,E1 -23305.053,E2 -23305.053} C_VEL
LIN {X 0,Y 164.038,Z 278.123,A -85,B 0,C 180,E1 -23308.773,E2 -23308.773} C_VEL
LIN {X 0,Y 165.523,Z 271.906,A -85,B 0,C 180,E1 -23312.434,E2 -23312.434} C_VEL
LIN {X 0,Y 167.598,Z 264.149,A -85,B 0,C 180,E1 -23316.018,E2 -23316.018} C_VEL
LIN {X 0,Y 170.248,Z 254.402,A -85,B 0,C 180,E1 -23319.505,E2 -23319.505} C_VEL
LIN {X 0,Y 172.729,Z 244.528,A -85,B 0,C 180,E1 -23322.287,E2 -23322.287} C_VEL
LIN {X 0,Y 175.247,Z 232.972,A -85,B 0,C 180,E1 -23324.813,E2 -23324.813} C_VEL
LIN {X 0,Y 177.344,Z 221.83,A -85,B 0,C 180,E1 -23326.698,E2 -23326.698} C_VEL
LIN {X 0,Y 179.238,Z 209.396,A -85,B 0,C 180,E1 -23328.282,E2 -23328.282} C_VEL
LIN {X 0,Y 180.698,Z 196.44,A -85,B 0,C 180,E1 -23329.427,E2 -23329.427} C_VEL
LIN {X 0,Y 181.567,Z 184.098,A -85,B 0,C 180,E1 -23330.124,E2 -23330.124} C_VEL
LIN {X 0,Y 184.165,Z 131.56,A -85,B 0,C 180,E1 -23332.032,E2 -23332.032} C_VEL
LIN {X 0,Y 179.921,Z 121.227,A -85,B 0,C 180,E1 -23333.316,E2 -23333.316} C_VEL
LIN {X 0,Y 171.868,Z 105.455,A -85,B 0,C 180,E1 -23335.789,E2 -23335.789} C_VEL
LIN {X 0,Y 166.092,Z 95.849,A -85,B 0,C 180,E1 -23337.665,E2 -23337.665} C_VEL
LIN {X 0,Y 164.605,Z 93.176,A -85,B 0,C 180,E1 -23338.187,E2 -23338.187} C_VEL
LIN {X 0,Y 164.364,Z 91.999,A -85,B 0,C 180,E1 -23338.406,E2 -23338.406} C_VEL
LIN {X 0,Y 164.378,Z 92.006,A -85,B 0,C 180,E1 -23341.227,E2 -23341.227} C_VEL
LIN {X 0,Y 164.341,Z 92.012,A -85,B 0,C 180,E1 -23346.778,E2 -23346.778} C_VEL
LIN {X 0,Y 164.31,Z 92.011,A -85,B 0,C 180,E1 -23349.912,E2 -23349.912} C_VEL
LIN {X 0,Y 164.31,Z 92.014,A -85,B 0,C 180,E1 -23353.352,E2 -23353.352} C_VEL
LIN {X 0,Y 164.296,Z 92.015,A -85,B 0,C 180,E1 -23356.809,E2 -23356.809} C_VEL
LIN {X 0,Y 164.3,Z 92.005,A -85,B 0,C 180,E1 -23360.351,E2 -23360.351} C_VEL
LIN {X 0,Y 164.333,Z 91.962,A -85,B 0,C 180,E1 -23364.349,E2 -23364.349} C_VEL
LIN {X 0,Y 164.393,Z 91.997,A -85,B 0,C 180,E1 -23369.134,E2 -23369.134} C_VEL
LIN {X 0,Y 164.42,Z 91.99,A -85,B 0,C 180,E1 -23374.694,E2 -23374.694} C_VEL
LIN {X 0,Y 164.488,Z 91.996,A -85,B 0,C 180,E1 -23380.051,E2 -23380.051} C_VEL
LIN {X 0,Y 164.527,Z 91.981,A -85,B 0,C 180,E1 -23385.149,E2 -23385.149} C_VEL
LIN {X 0,Y 164.771,Z 91.952,A -85,B 0,C 180,E1 -23390.176,E2 -23390.176} C_VEL
LIN {X 0,Y 164.834,Z 91.938,A -85,B 0,C 180,E1 -23392.651,E2 -23392.651} C_VEL
LIN {X 0,Y 165.051,Z 91.922,A -85,B 0,C 180,E1 -23397.559,E2 -23397.559} C_VEL
LIN {X 0,Y 165.298,Z 91.88,A -85,B 0,C 180,E1 -23399.999,E2 -23399.999} C_VEL
LIN {X 0,Y 164.765,Z 91.96,A -85,B 0,C 180,E1 -23404.893,E2 -23404.893} C_VEL
LIN {X 0,Y 164.832,Z 91.94,A -85,B 0,C 180,E1 -23407.348,E2 -23407.348} C_VEL
LIN {X 0,Y 164.705,Z 91.967,A -85,B 0,C 180,E1 -23411.06,E2 -23411.06} C_VEL
LIN {X 0,Y 164.485,Z 91.991,A -85,B 0,C 180,E1 -23417.402,E2 -23417.402} C_VEL
LIN {X 0,Y 164.475,Z 91.996,A -85,B 0,C 180,E1 -23419.988,E2 -23419.988} C_VEL
LIN {X 0,Y 164.388,Z 92.004,A -85,B 0,C 180,E1 -23426.128,E2 -23426.128} C_VEL
LIN {X 0,Y 164.378,Z 91.997,A -85,B 0,C 180,E1 -23431.227,E2 -23431.227} C_VEL
LIN {X 0,Y 164.296,Z 92.019,A -85,B 0,C 180,E1 -23436.789,E2 -23436.789} C_VEL
LIN {X 0,Y 164.292,Z 92.015,A -85,B 0,C 180,E1 -23439.915,E2 -23439.915} C_VEL
LIN {X 0,Y 164.293,Z 92.027,A -85,B 0,C 180,E1 -23444.894,E2 -23444.894} C_VEL
LIN {X 0,Y 165.381,Z 96.166,A -85,B 0,C 180,E1 -23447.407,E2 -23447.407} C_VEL
LIN {X 0,Y 171.83,Z 109.457,A -85,B 0,C 180,E1 -23449.639,E2 -23449.639} C_VEL
LIN {X 0,Y 177.205,Z 122.799,A -85,B 0,C 180,E1 -23451.448,E2 -23451.448} C_VEL
LIN {X 0,Y 180.135,Z 131.016,A -85,B 0,C 180,E1 -23452.419,E2 -23452.419} C_VEL
LIN {X 0,Y 182.743,Z 161.674,A -85,B 0,C 180,E1 -23454.3,E2 -23454.3} C_VEL
LIN {X 0,Y 180.659,Z 206.222,A -85,B 0,C 180,E1 -23456.003,E2 -23456.003} C_VEL
LIN {X 0,Y 179.339,Z 219.322,A -85,B 0,C 180,E1 -23456.893,E2 -23456.893} C_VEL
LIN {X 0,Y 177.513,Z 232.042,A -85,B 0,C 180,E1 -23458.192,E2 -23458.192} C_VEL
LIN {X 0,Y 175.206,Z 244.113,A -85,B 0,C 180,E1 -23459.906,E2 -23459.906} C_VEL
LIN {X 0,Y 172.597,Z 255.663,A -85,B 0,C 180,E1 -23462.077,E2 -23462.077} C_VEL
LIN {X 0,Y 170.051,Z 266.078,A -85,B 0,C 180,E1 -23464.609,E2 -23464.609} C_VEL
LIN {X 0,Y 168.874,Z 270.813,A -85,B 0,C 180,E1 -23465.999,E2 -23465.999} C_VEL
LIN {X 0,Y 167.108,Z 275.013,A -85,B 0,C 180,E1 -23467.313,E2 -23467.313} C_VEL
LIN {X 0,Y 160.832,Z 283.624,A -85,B 0,C 180,E1 -23470.42,E2 -23470.42} C_VEL
LIN {X 0,Y 157.786,Z 288.086,A -85,B 0,C 180,E1 -23472.495,E2 -23472.495} C_VEL
LIN {X 0,Y 156.932,Z 290.196,A -85,B 0,C 180,E1 -23473.653,E2 -23473.653} C_VEL
LIN {X 0,Y 155.811,Z 295.441,A -85,B 0,C 180,E1 -23476.965,E2 -23476.965} C_VEL
LIN {X 0,Y 155.176,Z 300.371,A -85,B 0,C 180,E1 -23480.878,E2 -23480.878} C_VEL
LIN {X 0,Y 155.087,Z 304.742,A -85,B 0,C 180,E1 -23485.531,E2 -23485.531} C_VEL
LIN {X 0,Y 155.304,Z 307.535,A -85,B 0,C 180,E1 -23489.999,E2 -23489.999} C_VEL
LIN {X 0,Y 155.021,Z 308.939,A -85,B 0,C 180,E1 -23494.144,E2 -23494.144} C_VEL
LIN {X 0,Y 154.972,Z 309.303,A -85,B 0,C 180,E1 -23497.818,E2 -23497.818} C_VEL
LIN {X 0,Y 155.347,Z 309.126,A -85,B 0,C 180,E1 -23500.425,E2 -23500.425} C_VEL
LIN {X 0,Y 156.824,Z 307.543,A -85,B 0,C 180,E1 -23505.597,E2 -23505.597} C_VEL
LIN {X 0,Y 159.784,Z 304.424,A -85,B 0,C 180,E1 -23510.601,E2 -23510.601} C_VEL
LIN {X 0,Y 162.792,Z 300.938,A -85,B 0,C 180,E1 -23514.212,E2 -23514.212} C_VEL
LIN {X 0,Y 166.259,Z 296.404,A -85,B 0,C 180,E1 -23517.708,E2 -23517.708} C_VEL
LIN {X 0,Y 171.288,Z 289.609,A -85,B 0,C 180,E1 -23521.542,E2 -23521.542} C_VEL
LIN {X 0,Y 176.304,Z 282.257,A -85,B 0,C 180,E1 -23524.613,E2 -23524.613} C_VEL
LIN {X 0,Y 181.79,Z 273.181,A -85,B 0,C 180,E1 -23527.508,E2 -23527.508} C_VEL
LIN {X 0,Y 186.268,Z 264.843,A -85,B 0,C 180,E1 -23529.545,E2 -23529.545} C_VEL
LIN {X 0,Y 191.031,Z 254.704,A -85,B 0,C 180,E1 -23531.468,E2 -23531.468} C_VEL
LIN {X 0,Y 195.568,Z 243.472,A -85,B 0,C 180,E1 -23533.061,E2 -23533.061} C_VEL
LIN {X 0,Y 199.706,Z 230.856,A -85,B 0,C 180,E1 -23534.38,E2 -23534.38} C_VEL
LIN {X 0,Y 202.787,Z 217.86,A -85,B 0,C 180,E1 -23535.359,E2 -23535.359} C_VEL
LIN {X 0,Y 204.961,Z 204.004,A -85,B 0,C 180,E1 -23536.06,E2 -23536.06} C_VEL
LIN {X 0,Y 207.283,Z 173.048,A -85,B 0,C 180,E1 -23537.048,E2 -23537.048} C_VEL
LIN {X 0,Y 206.889,Z 170.817,A -85,B 0,C 180,E1 -23537.319,E2 -23537.319} C_VEL
LIN {X 0,Y 202.559,Z 159.802,A -85,B 0,C 180,E1 -23539.649,E2 -23539.649} C_VEL
LIN {X 0,Y 198.269,Z 150.509,A -85,B 0,C 180,E1 -23542.116,E2 -23542.116} C_VEL
LIN {X 0,Y 193.52,Z 141.101,A -85,B 0,C 180,E1 -23545.14,E2 -23545.14} C_VEL
LIN {X 0,Y 189.877,Z 134.687,A -85,B 0,C 180,E1 -23547.749,E2 -23547.749} C_VEL
LIN {X 0,Y 187.247,Z 130.182,A -85,B 0,C 180,E1 -23549.854,E2 -23549.854} C_VEL
LIN {X 0,Y 183.645,Z 124.304,A -85,B 0,C 180,E1 -23553.143,E2 -23553.143} C_VEL
LIN {X 0,Y 180.005,Z 118.551,A -85,B 0,C 180,E1 -23557.224,E2 -23557.224} C_VEL
LIN {X 0,Y 177.527,Z 115.489,A -85,B 0,C 180,E1 -23560.716,E2 -23560.716} C_VEL
LIN {X 0,Y 175.581,Z 112.204,A -85,B 0,C 180,E1 -23564.711,E2 -23564.711} C_VEL
LIN {X 0,Y 175.268,Z 111.212,A -85,B 0,C 180,E1 -23565.681,E2 -23565.681} C_VEL
LIN {X 0,Y 173.716,Z 110.454,A -85,B 0,C 180,E1 -23573.029,E2 -23573.029} C_VEL
LIN {X 0,Y 175.321,Z 110.976,A -85,B 0,C 180,E1 -23581.149,E2 -23581.149} C_VEL
LIN {X 0,Y 175.664,Z 111.876,A -85,B 0,C 180,E1 -23582.15,E2 -23582.15} C_VEL
LIN {X 0,Y 177.178,Z 114.719,A -85,B 0,C 180,E1 -23585.406,E2 -23585.406} C_VEL
LIN {X 0,Y 179.621,Z 116.889,A -85,B 0,C 180,E1 -23588.916,E2 -23588.916} C_VEL
LIN {X 0,Y 181.627,Z 120.263,A -85,B 0,C 180,E1 -23591.403,E2 -23591.403} C_VEL
LIN {X 0,Y 183.685,Z 122.326,A -85,B 0,C 180,E1 -23593.457,E2 -23593.457} C_VEL
LIN {X 0,Y 186.472,Z 126.187,A -85,B 0,C 180,E1 -23596.003,E2 -23596.003} C_VEL
LIN {X 0,Y 190.771,Z 132.216,A -85,B 0,C 180,E1 -23599.364,E2 -23599.364} C_VEL
LIN {X 0,Y 194.271,Z 137.379,A -85,B 0,C 180,E1 -23601.757,E2 -23601.757} C_VEL
LIN {X 0,Y 199.118,Z 144.813,A -85,B 0,C 180,E1 -23604.671,E2 -23604.671} C_VEL
LIN {X 0,Y 204.835,Z 154.625,A -85,B 0,C 180,E1 -23607.733,E2 -23607.733} C_VEL
LIN {X 0,Y 208.126,Z 160.927,A -85,B 0,C 180,E1 -23609.352,E2 -23609.352} C_VEL
LIN {X 0,Y 205.827,Z 191.012,A -85,B 0,C 180,E1 -23610.328,E2 -23610.328} C_VEL
LIN {X 0,Y 203.733,Z 204.991,A -85,B 0,C 180,E1 -23611.115,E2 -23611.115} C_VEL
LIN {X 0,Y 200.924,Z 217.823,A -85,B 0,C 180,E1 -23612.238,E2 -23612.238} C_VEL
LIN {X 0,Y 197.34,Z 229.783,A -85,B 0,C 180,E1 -23613.648,E2 -23613.648} C_VEL
LIN {X 0,Y 193.089,Z 241.176,A -85,B 0,C 180,E1 -23615.427,E2 -23615.427} C_VEL
LIN {X 0,Y 188.357,Z 251.535,A -85,B 0,C 180,E1 -23617.546,E2 -23617.546} C_VEL
LIN {X 0,Y 183.428,Z 260.742,A -85,B 0,C 180,E1 -23619.979,E2 -23619.979} C_VEL
LIN {X 0,Y 178.838,Z 268.271,A -85,B 0,C 180,E1 -23622.538,E2 -23622.538} C_VEL
LIN {X 0,Y 173.824,Z 275.593,A -85,B 0,C 180,E1 -23625.779,E2 -23625.779} C_VEL
LIN {X 0,Y 170.055,Z 280.486,A -85,B 0,C 180,E1 -23628.606,E2 -23628.606} C_VEL
LIN {X 0,Y 166.047,Z 285.158,A -85,B 0,C 180,E1 -23632.142,E2 -23632.142} C_VEL
LIN {X 0,Y 162.646,Z 288.647,A -85,B 0,C 180,E1 -23635.825,E2 -23635.825} C_VEL
LIN {X 0,Y 160.73,Z 290.349,A -85,B 0,C 180,E1 -23638.353,E2 -23638.353} C_VEL
LIN {X 0,Y 158.185,Z 292.229,A -85,B 0,C 180,E1 -23642.697,E2 -23642.697} C_VEL
LIN {X 0,Y 156.649,Z 292.873,A -85,B 0,C 180,E1 -23646.186,E2 -23646.186} C_VEL
LIN {X 0,Y 155.842,Z 292.852,A -85,B 0,C 180,E1 -23648.853,E2 -23648.853} C_VEL
LIN {X 0,Y 155.213,Z 292.339,A -85,B 0,C 180,E1 -23651.969,E2 -23651.969} C_VEL
LIN {X 0,Y 154.781,Z 290.32,A -85,B 0,C 180,E1 -23656.879,E2 -23656.879} C_VEL
LIN {X 0,Y 155.078,Z 287.611,A -85,B 0,C 180,E1 -23660.874,E2 -23660.874} C_VEL
LIN {X 0,Y 155.816,Z 283.877,A -85,B 0,C 180,E1 -23664.825,E2 -23664.825} C_VEL
LIN {X 0,Y 156.878,Z 279.035,A -85,B 0,C 180,E1 -23668.717,E2 -23668.717} C_VEL
LIN {X 0,Y 158.391,Z 272.937,A -85,B 0,C 180,E1 -23672.544,E2 -23672.544} C_VEL
LIN {X 0,Y 160.513,Z 265.348,A -85,B 0,C 180,E1 -23676.285,E2 -23676.285} C_VEL
LIN {X 0,Y 162.738,Z 257.587,A -85,B 0,C 180,E1 -23679.321,E2 -23679.321} C_VEL
LIN {X 0,Y 165.274,Z 248.124,A -85,B 0,C 180,E1 -23682.277,E2 -23682.277} C_VEL
LIN {X 0,Y 167.882,Z 237.61,A -85,B 0,C 180,E1 -23684.858,E2 -23684.858} C_VEL
LIN {X 0,Y 170.221,Z 225.984,A -85,B 0,C 180,E1 -23687.109,E2 -23687.109} C_VEL
LIN {X 0,Y 172.385,Z 213.546,A -85,B 0,C 180,E1 -23688.882,E2 -23688.882} C_VEL
LIN {X 0,Y 174.109,Z 200.455,A -85,B 0,C 180,E1 -23690.221,E2 -23690.221} C_VEL
LIN {X 0,Y 175.155,Z 187.518,A -85,B 0,C 180,E1 -23691.093,E2 -23691.093} C_VEL
LIN {X 0,Y 177.901,Z 132.792,A -85,B 0,C 180,E1 -23693.175,E2 -23693.175} C_VEL
LIN {X 0,Y 172.916,Z 121.428,A -85,B 0,C 180,E1 -23694.761,E2 -23694.761} C_VEL
LIN {X 0,Y 165.358,Z 106.998,A -85,B 0,C 180,E1 -23697.256,E2 -23697.256} C_VEL
LIN {X 0,Y 159.022,Z 96.631,A -85,B 0,C 180,E1 -23699.496,E2 -23699.496} C_VEL
LIN {X 0,Y 157.568,Z 93.948,A -85,B 0,C 180,E1 -23700.063,E2 -23700.063} C_VEL
LIN {X 0,Y 157.363,Z 92.884,A -85,B 0,C 180,E1 -23700.257,E2 -23700.257} C_VEL
LIN {X 0,Y 157.3,Z 92.887,A -85,B 0,C 180,E1 -23706.463,E2 -23706.463} C_VEL
LIN {X 0,Y 157.218,Z 92.9,A -85,B 0,C 180,E1 -23712.109,E2 -23712.109} C_VEL
LIN {X 0,Y 157.215,Z 92.899,A -85,B 0,C 180,E1 -23717.889,E2 -23717.889} C_VEL
LIN {X 0,Y 157.271,Z 92.841,A -85,B 0,C 180,E1 -23723.551,E2 -23723.551} C_VEL
LIN {X 0,Y 157.296,Z 92.869,A -85,B 0,C 180,E1 -23728.096,E2 -23728.096} C_VEL
LIN {X 0,Y 157.325,Z 92.883,A -85,B 0,C 180,E1 -23733.466,E2 -23733.466} C_VEL
LIN {X 0,Y 157.398,Z 92.878,A -85,B 0,C 180,E1 -23739.667,E2 -23739.667} C_VEL
LIN {X 0,Y 157.457,Z 92.856,A -85,B 0,C 180,E1 -23744.466,E2 -23744.466} C_VEL
LIN {X 0,Y 157.693,Z 92.836,A -85,B 0,C 180,E1 -23749.73,E2 -23749.73} C_VEL
LIN {X 0,Y 157.771,Z 92.816,A -85,B 0,C 180,E1 -23752.32,E2 -23752.32} C_VEL
LIN {X 0,Y 158.26,Z 92.756,A -85,B 0,C 180,E1 -23759.999,E2 -23759.999} C_VEL
LIN {X 0,Y 157.769,Z 92.818,A -85,B 0,C 180,E1 -23767.679,E2 -23767.679} C_VEL
LIN {X 0,Y 157.64,Z 92.848,A -85,B 0,C 180,E1 -23771.236,E2 -23771.236} C_VEL
LIN {X 0,Y 157.444,Z 92.86,A -85,B 0,C 180,E1 -23775.535,E2 -23775.535} C_VEL
LIN {X 0,Y 157.37,Z 92.878,A -85,B 0,C 180,E1 -23780.932,E2 -23780.932} C_VEL
LIN {X 0,Y 157.311,Z 92.887,A -85,B 0,C 180,E1 -23786.68,E2 -23786.68} C_VEL
LIN {X 0,Y 157.277,Z 92.889,A -85,B 0,C 180,E1 -23792.426,E2 -23792.426} C_VEL
LIN {X 0,Y 157.27,Z 92.895,A -85,B 0,C 180,E1 -23796.449,E2 -23796.449} C_VEL
LIN {X 0,Y 157.212,Z 92.901,A -85,B 0,C 180,E1 -23802.11,E2 -23802.11} C_VEL
LIN {X 0,Y 157.259,Z 93.057,A -85,B 0,C 180,E1 -23803.716,E2 -23803.716} C_VEL
LIN {X 0,Y 157.96,Z 95.669,A -85,B 0,C 180,E1 -23805.387,E2 -23805.387} C_VEL
LIN {X 0,Y 160.361,Z 100.228,A -85,B 0,C 180,E1 -23806.313,E2 -23806.313} C_VEL
LIN {X 0,Y 166.737,Z 113.557,A -85,B 0,C 180,E1 -23808.659,E2 -23808.659} C_VEL
LIN {X 0,Y 171.707,Z 126.094,A -85,B 0,C 180,E1 -23810.442,E2 -23810.442} C_VEL
LIN {X 0,Y 174.176,Z 132.934,A -85,B 0,C 180,E1 -23811.308,E2 -23811.308} C_VEL
LIN {X 0,Y 176.576,Z 162.36,A -85,B 0,C 180,E1 -23813.193,E2 -23813.193} C_VEL
LIN {X 0,Y 174.458,Z 205.72,A -85,B 0,C 180,E1 -23814.897,E2 -23814.897} C_VEL
LIN {X 0,Y 173,Z 219.506,A -85,B 0,C 180,E1 -23815.866,E2 -23815.866} C_VEL
LIN {X 0,Y 171.102,Z 232.061,A -85,B 0,C 180,E1 -23817.201,E2 -23817.201} C_VEL
LIN {X 0,Y 168.708,Z 244.027,A -85,B 0,C 180,E1 -23818.967,E2 -23818.967} C_VEL
LIN {X 0,Y 165.978,Z 255.519,A -85,B 0,C 180,E1 -23821.206,E2 -23821.206} C_VEL
LIN {X 0,Y 163.317,Z 265.882,A -85,B 0,C 180,E1 -23823.826,E2 -23823.826} C_VEL
LIN {X 0,Y 161.122,Z 273.849,A -85,B 0,C 180,E1 -23826.348,E2 -23826.348} C_VEL
LIN {X 0,Y 159.15,Z 281.456,A -85,B 0,C 180,E1 -23829.311,E2 -23829.311} C_VEL
LIN {X 0,Y 157.186,Z 289.221,A -85,B 0,C 180,E1 -23833.104,E2 -23833.104} C_VEL
LIN {X 0,Y 156.932,Z 290.196,A -85,B 0,C 180,E1 -23833.653,E2 -23833.653} C_VEL
LIN {X 0,Y 155.559,Z 293.22,A -85,B 0,C 180,E1 -23835.447,E2 -23835.447} C_VEL
LIN {X 0,Y 151.91,Z 297.513,A -85,B 0,C 180,E1 -23838.491,E2 -23838.491} C_VEL
LIN {X 0,Y 148.671,Z 301.139,A -85,B 0,C 180,E1 -23841.802,E2 -23841.802} C_VEL
LIN {X 0,Y 147.974,Z 303.032,A -85,B 0,C 180,E1 -23843.951,E2 -23843.951} C_VEL
LIN {X 0,Y 148.032,Z 305.494,A -85,B 0,C 180,E1 -23847.278,E2 -23847.278} C_VEL
LIN {X 0,Y 148.216,Z 307.021,A -85,B 0,C 180,E1 -23849.999,E2 -23849.999} C_VEL
LIN {X 0,Y 147.945,Z 308.389,A -85,B 0,C 180,E1 -23853.984,E2 -23853.984} C_VEL
LIN {X 0,Y 147.932,Z 308.9,A -85,B 0,C 180,E1 -23858.193,E2 -23858.193} C_VEL
LIN {X 0,Y 148.329,Z 308.759,A -85,B 0,C 180,E1 -23860.924,E2 -23860.924} C_VEL
LIN {X 0,Y 148.988,Z 308.221,A -85,B 0,C 180,E1 -23863.641,E2 -23863.641} C_VEL
LIN {X 0,Y 149.963,Z 307.27,A -85,B 0,C 180,E1 -23866.33,E2 -23866.33} C_VEL
LIN {X 0,Y 153.117,Z 304.222,A -85,B 0,C 180,E1 -23871.542,E2 -23871.542} C_VEL
LIN {X 0,Y 156.311,Z 300.81,A -85,B 0,C 180,E1 -23875.285,E2 -23875.285} C_VEL
LIN {X 0,Y 159.98,Z 296.356,A -85,B 0,C 180,E1 -23878.896,E2 -23878.896} C_VEL
LIN {X 0,Y 165.267,Z 289.691,A -85,B 0,C 180,E1 -23882.832,E2 -23882.832} C_VEL
LIN {X 0,Y 170.515,Z 282.439,A -85,B 0,C 180,E1 -23885.967,E2 -23885.967} C_VEL
LIN {X 0,Y 176.226,Z 273.478,A -85,B 0,C 180,E1 -23888.91,E2 -23888.91} C_VEL
LIN {X 0,Y 180.385,Z 266.247,A -85,B 0,C 180,E1 -23890.737,E2 -23890.737} C_VEL
LIN {X 0,Y 183.656,Z 260.032,A -85,B 0,C 180,E1 -23892.041,E2 -23892.041} C_VEL
LIN {X 0,Y 188.133,Z 250.213,A -85,B 0,C 180,E1 -23893.716,E2 -23893.716} C_VEL
LIN {X 0,Y 192.883,Z 237.803,A -85,B 0,C 180,E1 -23895.275,E2 -23895.275} C_VEL
LIN {X 0,Y 196.692,Z 225.029,A -85,B 0,C 180,E1 -23896.449,E2 -23896.449} C_VEL
LIN {X 0,Y 199.47,Z 211.747,A -85,B 0,C 180,E1 -23897.295,E2 -23897.295} C_VEL
LIN {X 0,Y 201.182,Z 198.247,A -85,B 0,C 180,E1 -23897.853,E2 -23897.853} C_VEL
LIN {X 0,Y 202.926,Z 174.487,A -85,B 0,C 180,E1 -23898.604,E2 -23898.604} C_VEL
LIN {X 0,Y 198.776,Z 163.652,A -85,B 0,C 180,E1 -23901.012,E2 -23901.012} C_VEL
LIN {X 0,Y 194.767,Z 154.769,A -85,B 0,C 180,E1 -23903.491,E2 -23903.491} C_VEL
LIN {X 0,Y 190.536,Z 146.108,A -85,B 0,C 180,E1 -23906.408,E2 -23906.408} C_VEL
LIN {X 0,Y 187.291,Z 140.177,A -85,B 0,C 180,E1 -23908.908,E2 -23908.908} C_VEL
LIN {X 0,Y 184.873,Z 135.867,A -85,B 0,C 180,E1 -23910.988,E2 -23910.988} C_VEL
LIN {X 0,Y 181.715,Z 130.475,A -85,B 0,C 180,E1 -23914.083,E2 -23914.083} C_VEL
LIN {X 0,Y 178.419,Z 125.071,A -85,B 0,C 180,E1 -23918.032,E2 -23918.032} C_VEL
LIN {X 0,Y 176.207,Z 122.214,A -85,B 0,C 180,E1 -23921.393,E2 -23921.393} C_VEL
LIN {X 0,Y 174.344,Z 118.635,A -85,B 0,C 180,E1 -23925.672,E2 -23925.672} C_VEL
LIN {X 0,Y 174.045,Z 118.158,A -85,B 0,C 180,E1 -23926.575,E2 -23926.575} C_VEL
LIN {X 0,Y 172.845,Z 117.481,A -85,B 0,C 180,E1 -23932.994,E2 -23932.994} C_VEL
LIN {X 0,Y 174.375,Z 117.999,A -85,B 0,C 180,E1 -23940.993,E2 -23940.993} C_VEL
LIN {X 0,Y 175.565,Z 120.988,A -85,B 0,C 180,E1 -23944.111,E2 -23944.111} C_VEL
LIN {X 0,Y 178.253,Z 123.734,A -85,B 0,C 180,E1 -23948.36,E2 -23948.36} C_VEL
LIN {X 0,Y 180.216,Z 127.04,A -85,B 0,C 180,E1 -23950.905,E2 -23950.905} C_VEL
LIN {X 0,Y 182.062,Z 129.004,A -85,B 0,C 180,E1 -23952.834,E2 -23952.834} C_VEL
LIN {X 0,Y 184.802,Z 132.841,A -85,B 0,C 180,E1 -23955.439,E2 -23955.439} C_VEL
LIN {X 0,Y 188.697,Z 138.584,A -85,B 0,C 180,E1 -23958.633,E2 -23958.633} C_VEL
LIN {X 0,Y 193.16,Z 145.302,A -85,B 0,C 180,E1 -23961.766,E2 -23961.766} C_VEL
LIN {X 0,Y 198.48,Z 154.283,A -85,B 0,C 180,E1 -23965.017,E2 -23965.017} C_VEL
LIN {X 0,Y 202.939,Z 162.528,A -85,B 0,C 180,E1 -23967.455,E2 -23967.455} C_VEL
LIN {X 0,Y 203.705,Z 164.03,A -85,B 0,C 180,E1 -23967.854,E2 -23967.854} C_VEL
LIN {X 0,Y 201.449,Z 191.919,A -85,B 0,C 180,E1 -23968.774,E2 -23968.774} C_VEL
LIN {X 0,Y 199.287,Z 205.711,A -85,B 0,C 180,E1 -23969.563,E2 -23969.563} C_VEL
LIN {X 0,Y 196.57,Z 217.664,A -85,B 0,C 180,E1 -23970.602,E2 -23970.602} C_VEL
LIN {X 0,Y 192.771,Z 229.965,A -85,B 0,C 180,E1 -23972.045,E2 -23972.045} C_VEL
LIN {X 0,Y 188.182,Z 241.795,A -85,B 0,C 180,E1 -23973.9,E2 -23973.9} C_VEL
LIN {X 0,Y 183.403,Z 251.794,A -85,B 0,C 180,E1 -23975.953,E2 -23975.953} C_VEL
LIN {X 0,Y 178.785,Z 260.188,A -85,B 0,C 180,E1 -23978.17,E2 -23978.17} C_VEL
LIN {X 0,Y 173.914,Z 267.874,A -85,B 0,C 180,E1 -23980.739,E2 -23980.739} C_VEL
LIN {X 0,Y 168.566,Z 275.355,A -85,B 0,C 180,E1 -23984.013,E2 -23984.013} C_VEL
LIN {X 0,Y 164.573,Z 280.355,A -85,B 0,C 180,E1 -23986.901,E2 -23986.901} C_VEL
LIN {X 0,Y 160.258,Z 285.147,A -85,B 0,C 180,E1 -23990.516,E2 -23990.516} C_VEL
LIN {X 0,Y 156.55,Z 288.745,A -85,B 0,C 180,E1 -23994.297,E2 -23994.297} C_VEL
LIN {X 0,Y 154.46,Z 290.535,A -85,B 0,C 180,E1 -23996.908,E2 -23996.908} C_VEL
LIN {X 0,Y 151.393,Z 292.644,A -85,B 0,C 180,E1 -24001.889,E2 -24001.889} C_VEL
LIN {X 0,Y 149.949,Z 293.245,A -85,B 0,C 180,E1 -24005.051,E2 -24005.051} C_VEL
LIN {X 0,Y 149.009,Z 293.273,A -85,B 0,C 180,E1 -24007.833,E2 -24007.833} C_VEL
LIN {X 0,Y 148.164,Z 292.709,A -85,B 0,C 180,E1 -24011.567,E2 -24011.567} C_VEL
LIN {X 0,Y 147.696,Z 290.927,A -85,B 0,C 180,E1 -24016.237,E2 -24016.237} C_VEL
LIN {X 0,Y 147.923,Z 288.315,A -85,B 0,C 180,E1 -24020.429,E2 -24020.429} C_VEL
LIN {X 0,Y 148.636,Z 284.682,A -85,B 0,C 180,E1 -24024.575,E2 -24024.575} C_VEL
LIN {X 0,Y 149.719,Z 279.947,A -85,B 0,C 180,E1 -24028.656,E2 -24028.656} C_VEL
LIN {X 0,Y 151.582,Z 272.84,A -85,B 0,C 180,E1 -24033.323,E2 -24033.323} C_VEL
LIN {X 0,Y 153.855,Z 265.134,A -85,B 0,C 180,E1 -24037.217,E2 -24037.217} C_VEL
LIN {X 0,Y 156.739,Z 255.435,A -85,B 0,C 180,E1 -24040.987,E2 -24040.987} C_VEL
LIN {X 0,Y 159.404,Z 245.793,A -85,B 0,C 180,E1 -24043.929,E2 -24043.929} C_VEL
LIN {X 0,Y 161.911,Z 235.584,A -85,B 0,C 180,E1 -24046.389,E2 -24046.389} C_VEL
LIN {X 0,Y 164.134,Z 224.897,A -85,B 0,C 180,E1 -24048.409,E2 -24048.409} C_VEL
LIN {X 0,Y 166.235,Z 213.141,A -85,B 0,C 180,E1 -24050.091,E2 -24050.091} C_VEL
LIN {X 0,Y 167.939,Z 200.541,A -85,B 0,C 180,E1 -24051.4,E2 -24051.4} C_VEL
LIN {X 0,Y 169.012,Z 188.286,A -85,B 0,C 180,E1 -24052.245,E2 -24052.245} C_VEL
LIN {X 0,Y 171.824,Z 134.659,A -85,B 0,C 180,E1 -24054.344,E2 -24054.344} C_VEL
LIN {X 0,Y 167.119,Z 124.142,A -85,B 0,C 180,E1 -24055.933,E2 -24055.933} C_VEL
LIN {X 0,Y 160.461,Z 111.272,A -85,B 0,C 180,E1 -24058.282,E2 -24058.282} C_VEL
LIN {X 0,Y 154.267,Z 101.02,A -85,B 0,C 180,E1 -24060.62,E2 -24060.62} C_VEL
LIN {X 0,Y 152.396,Z 97.969,A -85,B 0,C 180,E1 -24061.376,E2 -24061.376} C_VEL
LIN {X 0,Y 150.665,Z 95.429,A -85,B 0,C 180,E1 -24062.081,E2 -24062.081} C_VEL
LIN {X 0,Y 150.25,Z 93.752,A -85,B 0,C 180,E1 -24062.371,E2 -24062.371} C_VEL
LIN {X 0,Y 150.22,Z 93.773,A -85,B 0,C 180,E1 -24067.461,E2 -24067.461} C_VEL
LIN {X 0,Y 150.161,Z 93.777,A -85,B 0,C 180,E1 -24071.508,E2 -24071.508} C_VEL
LIN {X 0,Y 150.14,Z 93.772,A -85,B 0,C 180,E1 -24075.399,E2 -24075.399} C_VEL
LIN {X 0,Y 150.155,Z 93.775,A -85,B 0,C 180,E1 -24079.059,E2 -24079.059} C_VEL
LIN {X 0,Y 150.183,Z 93.728,A -85,B 0,C 180,E1 -24082.708,E2 -24082.708} C_VEL
LIN {X 0,Y 150.218,Z 93.74,A -85,B 0,C 180,E1 -24087.368,E2 -24087.368} C_VEL
LIN {X 0,Y 150.248,Z 93.767,A -85,B 0,C 180,E1 -24092.718,E2 -24092.718} C_VEL
LIN {X 0,Y 150.355,Z 93.756,A -85,B 0,C 180,E1 -24099.207,E2 -24099.207} C_VEL
LIN {X 0,Y 150.364,Z 93.738,A -85,B 0,C 180,E1 -24103.713,E2 -24103.713} C_VEL
LIN {X 0,Y 150.615,Z 93.721,A -85,B 0,C 180,E1 -24109.242,E2 -24109.242} C_VEL
LIN {X 0,Y 150.708,Z 93.695,A -85,B 0,C 180,E1 -24111.957,E2 -24111.957} C_VEL
LIN {X 0,Y 151.221,Z 93.632,A -85,B 0,C 180,E1 -24119.999,E2 -24119.999} C_VEL
LIN {X 0,Y 150.706,Z 93.697,A -85,B 0,C 180,E1 -24128.042,E2 -24128.042} C_VEL
LIN {X 0,Y 150.58,Z 93.728,A -85,B 0,C 180,E1 -24131.437,E2 -24131.437} C_VEL
LIN {X 0,Y 150.355,Z 93.744,A -85,B 0,C 180,E1 -24136.287,E2 -24136.287} C_VEL
LIN {X 0,Y 150.352,Z 93.753,A -85,B 0,C 180,E1 -24140.79,E2 -24140.79} C_VEL
LIN {X 0,Y 150.243,Z 93.768,A -85,B 0,C 180,E1 -24147.279,E2 -24147.279} C_VEL
LIN {X 0,Y 150.217,Z 93.77,A -85,B 0,C 180,E1 -24152.632,E2 -24152.632} C_VEL
LIN {X 0,Y 150.174,Z 93.778,A -85,B 0,C 180,E1 -24157.472,E2 -24157.472} C_VEL
LIN {X 0,Y 150.213,Z 93.897,A -85,B 0,C 180,E1 -24162.279,E2 -24162.279} C_VEL
LIN {X 0,Y 150.525,Z 95.12,A -85,B 0,C 180,E1 -24163.094,E2 -24163.094} C_VEL
LIN {X 0,Y 152.747,Z 99.348,A -85,B 0,C 180,E1 -24164.057,E2 -24164.057} C_VEL
LIN {X 0,Y 158.425,Z 110.518,A -85,B 0,C 180,E1 -24166.362,E2 -24166.362} C_VEL
LIN {X 0,Y 162.84,Z 120.264,A -85,B 0,C 180,E1 -24168.057,E2 -24168.057} C_VEL
LIN {X 0,Y 168.313,Z 135.163,A -85,B 0,C 180,E1 -24170.14,E2 -24170.14} C_VEL
LIN {X 0,Y 170.491,Z 163.187,A -85,B 0,C 180,E1 -24172.015,E2 -24172.015} C_VEL
LIN {X 0,Y 168.241,Z 206.052,A -85,B 0,C 180,E1 -24173.756,E2 -24173.756} C_VEL
LIN {X 0,Y 166.721,Z 219.689,A -85,B 0,C 180,E1 -24174.76,E2 -24174.76} C_VEL
LIN {X 0,Y 164.747,Z 232.061,A -85,B 0,C 180,E1 -24176.134,E2 -24176.134} C_VEL
LIN {X 0,Y 162.258,Z 243.94,A -85,B 0,C 180,E1 -24177.953,E2 -24177.953} C_VEL
LIN {X 0,Y 159.405,Z 255.375,A -85,B 0,C 180,E1 -24180.263,E2 -24180.263} C_VEL
LIN {X 0,Y 156.622,Z 265.684,A -85,B 0,C 180,E1 -24182.977,E2 -24182.977} C_VEL
LIN {X 0,Y 154.173,Z 274.109,A -85,B 0,C 180,E1 -24185.777,E2 -24185.777} C_VEL
LIN {X 0,Y 152.048,Z 281.9,A -85,B 0,C 180,E1 -24189.008,E2 -24189.008} C_VEL
LIN {X 0,Y 149.918,Z 289.989,A -85,B 0,C 180,E1 -24193.26,E2 -24193.26} C_VEL
LIN {X 0,Y 148.535,Z 296.514,A -85,B 0,C 180,E1 -24197.706,E2 -24197.706} C_VEL
LIN {X 0,Y 148.006,Z 301.12,A -85,B 0,C 180,E1 -24201.809,E2 -24201.809} C_VEL
LIN {X 0,Y 147.974,Z 303.032,A -85,B 0,C 180,E1 -24203.951,E2 -24203.951} C_VEL
LIN {X 0,Y 147.319,Z 304.707,A -85,B 0,C 180,E1 -24206.134,E2 -24206.134} C_VEL
LIN {X 0,Y 145.721,Z 306.032,A -85,B 0,C 180,E1 -24208.317,E2 -24208.317} C_VEL
LIN {X 0,Y 141.933,Z 307.735,A -85,B 0,C 180,E1 -24212.84,E2 -24212.84} C_VEL
LIN {X 0,Y 140.861,Z 308.173,A -85,B 0,C 180,E1 -24215.245,E2 -24215.245} C_VEL
LIN {X 0,Y 140.771,Z 308.262,A -85,B 0,C 180,E1 -24216.063,E2 -24216.063} C_VEL
LIN {X 0,Y 141.336,Z 308.388,A -85,B 0,C 180,E1 -24221.472,E2 -24221.472} C_VEL
LIN {X 0,Y 142.073,Z 307.902,A -85,B 0,C 180,E1 -24224.319,E2 -24224.319} C_VEL
LIN {X 0,Y 143.129,Z 307.001,A -85,B 0,C 180,E1 -24227.133,E2 -24227.133} C_VEL
LIN {X 0,Y 146.498,Z 304.022,A -85,B 0,C 180,E1 -24232.567,E2 -24232.567} C_VEL
LIN {X 0,Y 149.892,Z 300.684,A -85,B 0,C 180,E1 -24236.45,E2 -24236.45} C_VEL
LIN {X 0,Y 153.795,Z 296.309,A -85,B 0,C 180,E1 -24240.175,E2 -24240.175} C_VEL
LIN {X 0,Y 159.352,Z 289.763,A -85,B 0,C 180,E1 -24244.215,E2 -24244.215} C_VEL
LIN {X 0,Y 164.835,Z 282.621,A -85,B 0,C 180,E1 -24247.413,E2 -24247.413} C_VEL
LIN {X 0,Y 170.775,Z 273.774,A -85,B 0,C 180,E1 -24250.402,E2 -24250.402} C_VEL
LIN {X 0,Y 175.081,Z 266.679,A -85,B 0,C 180,E1 -24252.249,E2 -24252.249} C_VEL
LIN {X 0,Y 179.061,Z 259.466,A -85,B 0,C 180,E1 -24253.769,E2 -24253.769} C_VEL
LIN {X 0,Y 183.095,Z 250.943,A -85,B 0,C 180,E1 -24255.243,E2 -24255.243} C_VEL
LIN {X 0,Y 187.364,Z 240.626,A -85,B 0,C 180,E1 -24256.614,E2 -24256.614} C_VEL
LIN {X 0,Y 191.529,Z 228.027,A -85,B 0,C 180,E1 -24257.842,E2 -24257.842} C_VEL
LIN {X 0,Y 194.651,Z 214.852,A -85,B 0,C 180,E1 -24258.79,E2 -24258.79} C_VEL
LIN {X 0,Y 196.708,Z 201.838,A -85,B 0,C 180,E1 -24259.382,E2 -24259.382} C_VEL
LIN {X 0,Y 198.668,Z 177.094,A -85,B 0,C 180,E1 -24260.186,E2 -24260.186} C_VEL
LIN {X 0,Y 194.843,Z 166.865,A -85,B 0,C 180,E1 -24262.598,E2 -24262.598} C_VEL
LIN {X 0,Y 190.009,Z 156.025,A -85,B 0,C 180,E1 -24265.911,E2 -24265.911} C_VEL
LIN {X 0,Y 185.993,Z 147.803,A -85,B 0,C 180,E1 -24269.073,E2 -24269.073} C_VEL
LIN {X 0,Y 182.887,Z 142.121,A -85,B 0,C 180,E1 -24271.847,E2 -24271.847} C_VEL
LIN {X 0,Y 179.926,Z 136.79,A -85,B 0,C 180,E1 -24274.941,E2 -24274.941} C_VEL
LIN {X 0,Y 176.888,Z 131.617,A -85,B 0,C 180,E1 -24278.834,E2 -24278.834} C_VEL
LIN {X 0,Y 175.031,Z 129.066,A -85,B 0,C 180,E1 -24281.86,E2 -24281.86} C_VEL
LIN {X 0,Y 173.159,Z 125.196,A -85,B 0,C 180,E1 -24286.58,E2 -24286.58} C_VEL
LIN {X 0,Y 171.967,Z 124.529,A -85,B 0,C 180,E1 -24292.958,E2 -24292.958} C_VEL
LIN {X 0,Y 173.3,Z 124.969,A -85,B 0,C 180,E1 -24300.5,E2 -24300.5} C_VEL
LIN {X 0,Y 174.561,Z 128.02,A -85,B 0,C 180,E1 -24303.92,E2 -24303.92} C_VEL
LIN {X 0,Y 176.907,Z 130.567,A -85,B 0,C 180,E1 -24307.796,E2 -24307.796} C_VEL
LIN {X 0,Y 178.9,Z 133.916,A -85,B 0,C 180,E1 -24310.494,E2 -24310.494} C_VEL
LIN {X 0,Y 180.374,Z 135.562,A -85,B 0,C 180,E1 -24312.107,E2 -24312.107} C_VEL
LIN {X 0,Y 183.687,Z 140.472,A -85,B 0,C 180,E1 -24315.376,E2 -24315.376} C_VEL
LIN {X 0,Y 186.879,Z 145.334,A -85,B 0,C 180,E1 -24318.067,E2 -24318.067} C_VEL
LIN {X 0,Y 190.703,Z 151.32,A -85,B 0,C 180,E1 -24320.884,E2 -24320.884} C_VEL
LIN {X 0,Y 194.916,Z 158.623,A -85,B 0,C 180,E1 -24323.64,E2 -24323.64} C_VEL
LIN {X 0,Y 199.311,Z 166.974,A -85,B 0,C 180,E1 -24326.219,E2 -24326.219} C_VEL
LIN {X 0,Y 199.462,Z 167.276,A -85,B 0,C 180,E1 -24326.304,E2 -24326.304} C_VEL
LIN {X 0,Y 197.288,Z 192.484,A -85,B 0,C 180,E1 -24327.132,E2 -24327.132} C_VEL
LIN {X 0,Y 195.095,Z 205.954,A -85,B 0,C 180,E1 -24327.901,E2 -24327.901} C_VEL
LIN {X 0,Y 192.247,Z 218.036,A -85,B 0,C 180,E1 -24328.947,E2 -24328.947} C_VEL
LIN {X 0,Y 188.362,Z 230.176,A -85,B 0,C 180,E1 -24330.367,E2 -24330.367} C_VEL
LIN {X 0,Y 183.717,Z 241.779,A -85,B 0,C 180,E1 -24332.181,E2 -24332.181} C_VEL
LIN {X 0,Y 178.61,Z 252.061,A -85,B 0,C 180,E1 -24334.28,E2 -24334.28} C_VEL
LIN {X 0,Y 173.162,Z 261.476,A -85,B 0,C 180,E1 -24336.818,E2 -24336.818} C_VEL
LIN {X 0,Y 168.188,Z 268.87,A -85,B 0,C 180,E1 -24339.373,E2 -24339.373} C_VEL
LIN {X 0,Y 162.613,Z 276.234,A -85,B 0,C 180,E1 -24342.718,E2 -24342.718} C_VEL
LIN {X 0,Y 157.631,Z 282.012,A -85,B 0,C 180,E1 -24346.287,E2 -24346.287} C_VEL
LIN {X 0,Y 153.195,Z 286.493,A -85,B 0,C 180,E1 -24350.04,E2 -24350.04} C_VEL
LIN {X 0,Y 150.61,Z 288.832,A -85,B 0,C 180,E1 -24352.655,E2 -24352.655} C_VEL
LIN {X 0,Y 148.294,Z 290.713,A -85,B 0,C 180,E1 -24355.341,E2 -24355.341} C_VEL
LIN {X 0,Y 146.324,Z 292.091,A -85,B 0,C 180,E1 -24358.108,E2 -24358.108} C_VEL
LIN {X 0,Y 144.655,Z 293.055,A -85,B 0,C 180,E1 -24360.99,E2 -24360.99} C_VEL
LIN {X 0,Y 143.294,Z 293.588,A -85,B 0,C 180,E1 -24363.807,E2 -24363.807} C_VEL
LIN {X 0,Y 142.211,Z 293.694,A -85,B 0,C 180,E1 -24366.713,E2 -24366.713} C_VEL
LIN {X 0,Y 141.157,Z 293.087,A -85,B 0,C 180,E1 -24371.084,E2 -24371.084} C_VEL
LIN {X 0,Y 140.641,Z 291.522,A -85,B 0,C 180,E1 -24375.532,E2 -24375.532} C_VEL
LIN {X 0,Y 140.769,Z 288.999,A -85,B 0,C 180,E1 -24379.938,E2 -24379.938} C_VEL
LIN {X 0,Y 141.471,Z 285.463,A -85,B 0,C 180,E1 -24384.299,E2 -24384.299} C_VEL
LIN {X 0,Y 142.564,Z 280.842,A -85,B 0,C 180,E1 -24388.589,E2 -24388.589} C_VEL
LIN {X 0,Y 144.454,Z 273.861,A -85,B 0,C 180,E1 -24393.488,E2 -24393.488} C_VEL
LIN {X 0,Y 146.782,Z 266.304,A -85,B 0,C 180,E1 -24397.567,E2 -24397.567} C_VEL
LIN {X 0,Y 149.218,Z 258.582,A -85,B 0,C 180,E1 -24400.86,E2 -24400.86} C_VEL
LIN {X 0,Y 151.936,Z 249.419,A -85,B 0,C 180,E1 -24403.981,E2 -24403.981} C_VEL
LIN {X 0,Y 154.85,Z 238.733,A -85,B 0,C 180,E1 -24406.819,E2 -24406.819} C_VEL
LIN {X 0,Y 157.417,Z 227.19,A -85,B 0,C 180,E1 -24409.225,E2 -24409.225} C_VEL
LIN {X 0,Y 159.807,Z 214.921,A -85,B 0,C 180,E1 -24411.105,E2 -24411.105} C_VEL
LIN {X 0,Y 161.765,Z 201.296,A -85,B 0,C 180,E1 -24412.596,E2 -24412.596} C_VEL
LIN {X 0,Y 162.924,Z 188.875,A -85,B 0,C 180,E1 -24413.489,E2 -24413.489} C_VEL
LIN {X 0,Y 165.8,Z 136.58,A -85,B 0,C 180,E1 -24415.596,E2 -24415.596} C_VEL
LIN {X 0,Y 160.458,Z 124.814,A -85,B 0,C 180,E1 -24417.537,E2 -24417.537} C_VEL
LIN {X 0,Y 154.399,Z 113.292,A -85,B 0,C 180,E1 -24419.855,E2 -24419.855} C_VEL
LIN {X 0,Y 147.999,Z 102.897,A -85,B 0,C 180,E1 -24422.485,E2 -24422.485} C_VEL
LIN {X 0,Y 145.642,Z 99.199,A -85,B 0,C 180,E1 -24423.529,E2 -24423.529} C_VEL
LIN {X 0,Y 143.778,Z 96.751,A -85,B 0,C 180,E1 -24424.359,E2 -24424.359} C_VEL
LIN {X 0,Y 143.15,Z 94.633,A -85,B 0,C 180,E1 -24424.781,E2 -24424.781} C_VEL
LIN {X 0,Y 143.082,Z 94.654,A -85,B 0,C 180,E1 -24429.684,E2 -24429.684} C_VEL
LIN {X 0,Y 143.07,Z 94.659,A -85,B 0,C 180,E1 -24433.451,E2 -24433.451} C_VEL
LIN {X 0,Y 143.072,Z 94.661,A -85,B 0,C 180,E1 -24437.464,E2 -24437.464} C_VEL
LIN {X 0,Y 143.081,Z 94.621,A -85,B 0,C 180,E1 -24441.806,E2 -24441.806} C_VEL
LIN {X 0,Y 143.185,Z 94.612,A -85,B 0,C 180,E1 -24447.321,E2 -24447.321} C_VEL
LIN {X 0,Y 143.194,Z 94.648,A -85,B 0,C 180,E1 -24452.063,E2 -24452.063} C_VEL
LIN {X 0,Y 143.281,Z 94.636,A -85,B 0,C 180,E1 -24458.745,E2 -24458.745} C_VEL
LIN {X 0,Y 143.304,Z 94.618,A -85,B 0,C 180,E1 -24462.886,E2 -24462.886} C_VEL
LIN {X 0,Y 143.541,Z 94.602,A -85,B 0,C 180,E1 -24468.705,E2 -24468.705} C_VEL
LIN {X 0,Y 143.63,Z 94.577,A -85,B 0,C 180,E1 -24471.558,E2 -24471.558} C_VEL
LIN {X 0,Y 144.179,Z 94.508,A -85,B 0,C 180,E1 -24479.999,E2 -24479.999} C_VEL
LIN {X 0,Y 143.628,Z 94.579,A -85,B 0,C 180,E1 -24488.441,E2 -24488.441} C_VEL
LIN {X 0,Y 143.507,Z 94.61,A -85,B 0,C 180,E1 -24491.628,E2 -24491.628} C_VEL
LIN {X 0,Y 143.298,Z 94.627,A -85,B 0,C 180,E1 -24497.113,E2 -24497.113} C_VEL
LIN {X 0,Y 143.278,Z 94.633,A -85,B 0,C 180,E1 -24501.252,E2 -24501.252} C_VEL
LIN {X 0,Y 143.19,Z 94.646,A -85,B 0,C 180,E1 -24507.935,E2 -24507.935} C_VEL
LIN {X 0,Y 143.166,Z 94.651,A -85,B 0,C 180,E1 -24513.432,E2 -24513.432} C_VEL
LIN {X 0,Y 143.062,Z 94.659,A -85,B 0,C 180,E1 -24519.689,E2 -24519.689} C_VEL
LIN {X 0,Y 143.12,Z 94.855,A -85,B 0,C 180,E1 -24520.499,E2 -24520.499} C_VEL
LIN {X 0,Y 144.151,Z 97.574,A -85,B 0,C 180,E1 -24521.063,E2 -24521.063} C_VEL
LIN {X 0,Y 146.293,Z 100.341,A -85,B 0,C 180,E1 -24522.007,E2 -24522.007} C_VEL
LIN {X 0,Y 151.856,Z 111.066,A -85,B 0,C 180,E1 -24524.491,E2 -24524.491} C_VEL
LIN {X 0,Y 156.788,Z 121.795,A -85,B 0,C 180,E1 -24526.551,E2 -24526.551} C_VEL
LIN {X 0,Y 161.819,Z 135.399,A -85,B 0,C 180,E1 -24528.617,E2 -24528.617} C_VEL
LIN {X 0,Y 162.557,Z 137.654,A -85,B 0,C 180,E1 -24528.92,E2 -24528.92} C_VEL
LIN {X 0,Y 164.488,Z 164.037,A -85,B 0,C 180,E1 -24530.757,E2 -24530.757} C_VEL
LIN {X 0,Y 162.194,Z 205.232,A -85,B 0,C 180,E1 -24532.463,E2 -24532.463} C_VEL
LIN {X 0,Y 160.622,Z 219.072,A -85,B 0,C 180,E1 -24533.501,E2 -24533.501} C_VEL
LIN {X 0,Y 158.661,Z 230.992,A -85,B 0,C 180,E1 -24534.84,E2 -24534.84} C_VEL
LIN {X 0,Y 156.249,Z 242.241,A -85,B 0,C 180,E1 -24536.564,E2 -24536.564} C_VEL
LIN {X 0,Y 153.167,Z 253.899,A -85,B 0,C 180,E1 -24538.921,E2 -24538.921} C_VEL
LIN {X 0,Y 150.545,Z 263.347,A -85,B 0,C 180,E1 -24541.411,E2 -24541.411} C_VEL
LIN {X 0,Y 148.304,Z 271.236,A -85,B 0,C 180,E1 -24544,E2 -24544} C_VEL
LIN {X 0,Y 146.211,Z 277.757,A -85,B 0,C 180,E1 -24546.551,E2 -24546.551} C_VEL
LIN {X 0,Y 144.206,Z 285.014,A -85,B 0,C 180,E1 -24550.052,E2 -24550.052} C_VEL
LIN {X 0,Y 142.354,Z 291.923,A -85,B 0,C 180,E1 -24554.243,E2 -24554.243} C_VEL
LIN {X 0,Y 141.294,Z 297.443,A -85,B 0,C 180,E1 -24558.523,E2 -24558.523} C_VEL
LIN {X 0,Y 140.9,Z 301.741,A -85,B 0,C 180,E1 -24562.836,E2 -24562.836} C_VEL
LIN {X 0,Y 140.938,Z 304.926,A -85,B 0,C 180,E1 -24567.141,E2 -24567.141} C_VEL
LIN {X 0,Y 141.13,Z 306.49,A -85,B 0,C 180,E1 -24569.999,E2 -24569.999} C_VEL
LIN {X 0,Y 140.869,Z 307.825,A -85,B 0,C 180,E1 -24573.802,E2 -24573.802} C_VEL
LIN {X 0,Y 140.771,Z 308.262,A -85,B 0,C 180,E1 -24576.063,E2 -24576.063} C_VEL
LIN {X 0,Y 140.182,Z 308.466,A -85,B 0,C 180,E1 -24578.464,E2 -24578.464} C_VEL
LIN {X 0,Y 137.903,Z 308.142,A -85,B 0,C 180,E1 -24582.448,E2 -24582.448} C_VEL
LIN {X 0,Y 136.326,Z 307.22,A -85,B 0,C 180,E1 -24586.526,E2 -24586.526} C_VEL
LIN {X 0,Y 136.837,Z 306.317,A -85,B 0,C 180,E1 -24588.966,E2 -24588.966} C_VEL
LIN {X 0,Y 139.936,Z 303.823,A -85,B 0,C 180,E1 -24593.688,E2 -24593.688} C_VEL
LIN {X 0,Y 143.524,Z 300.558,A -85,B 0,C 180,E1 -24597.721,E2 -24597.721} C_VEL
LIN {X 0,Y 147.693,Z 296.261,A -85,B 0,C 180,E1 -24601.562,E2 -24601.562} C_VEL
LIN {X 0,Y 153.54,Z 289.806,A -85,B 0,C 180,E1 -24605.703,E2 -24605.703} C_VEL
LIN {X 0,Y 159.269,Z 282.806,A -85,B 0,C 180,E1 -24608.961,E2 -24608.961} C_VEL
LIN {X 0,Y 165.447,Z 274.086,A -85,B 0,C 180,E1 -24611.992,E2 -24611.992} C_VEL
LIN {X 0,Y 169.91,Z 267.134,A -85,B 0,C 180,E1 -24613.853,E2 -24613.853} C_VEL
LIN {X 0,Y 175.702,Z 256.612,A -85,B 0,C 180,E1 -24616.052,E2 -24616.052} C_VEL
LIN {X 0,Y 180.689,Z 246.19,A -85,B 0,C 180,E1 -24617.646,E2 -24617.646} C_VEL
LIN {X 0,Y 185.188,Z 234.747,A -85,B 0,C 180,E1 -24618.96,E2 -24618.96} C_VEL
LIN {X 0,Y 188.872,Z 222.331,A -85,B 0,C 180,E1 -24620.021,E2 -24620.021} C_VEL
LIN {X 0,Y 191.6,Z 209.616,A -85,B 0,C 180,E1 -24620.775,E2 -24620.775} C_VEL
LIN {X 0,Y 193.27,Z 196.525,A -85,B 0,C 180,E1 -24621.29,E2 -24621.29} C_VEL
LIN {X 0,Y 194.567,Z 179.829,A -85,B 0,C 180,E1 -24621.831,E2 -24621.831} C_VEL
LIN {X 0,Y 191.694,Z 171.806,A -85,B 0,C 180,E1 -24623.796,E2 -24623.796} C_VEL
LIN {X 0,Y 187.35,Z 161.52,A -85,B 0,C 180,E1 -24627.013,E2 -24627.013} C_VEL
LIN {X 0,Y 183.625,Z 153.508,A -85,B 0,C 180,E1 -24630.162,E2 -24630.162} C_VEL
LIN {X 0,Y 180.856,Z 148.217,A -85,B 0,C 180,E1 -24632.813,E2 -24632.813} C_VEL
LIN {X 0,Y 178.099,Z 142.98,A -85,B 0,C 180,E1 -24635.91,E2 -24635.91} C_VEL
LIN {X 0,Y 175.491,Z 138.269,A -85,B 0,C 180,E1 -24639.52,E2 -24639.52} C_VEL
LIN {X 0,Y 173.762,Z 135.793,A -85,B 0,C 180,E1 -24642.536,E2 -24642.536} C_VEL
LIN {X 0,Y 172.131,Z 132.172,A -85,B 0,C 180,E1 -24647.007,E2 -24647.007} C_VEL
LIN {X 0,Y 171.09,Z 131.577,A -85,B 0,C 180,E1 -24652.922,E2 -24652.922} C_VEL
LIN {X 0,Y 172.241,Z 131.917,A -85,B 0,C 180,E1 -24660.001,E2 -24660.001} C_VEL
LIN {X 0,Y 173.743,Z 135.362,A -85,B 0,C 180,E1 -24664.114,E2 -24664.114} C_VEL
LIN {X 0,Y 175.508,Z 137.246,A -85,B 0,C 180,E1 -24667.105,E2 -24667.105} C_VEL
LIN {X 0,Y 177.765,Z 140.972,A -85,B 0,C 180,E1 -24670.277,E2 -24670.277} C_VEL
LIN {X 0,Y 178.899,Z 142.43,A -85,B 0,C 180,E1 -24671.58,E2 -24671.58} C_VEL
LIN {X 0,Y 181.786,Z 146.859,A -85,B 0,C 180,E1 -24674.573,E2 -24674.573} C_VEL
LIN {X 0,Y 184.495,Z 151.086,A -85,B 0,C 180,E1 -24676.996,E2 -24676.996} C_VEL
LIN {X 0,Y 188.372,Z 157.455,A -85,B 0,C 180,E1 -24680.036,E2 -24680.036} C_VEL
LIN {X 0,Y 192.375,Z 164.727,A -85,B 0,C 180,E1 -24682.814,E2 -24682.814} C_VEL
LIN {X 0,Y 195.294,Z 170.337,A -85,B 0,C 180,E1 -24684.639,E2 -24684.639} C_VEL
LIN {X 0,Y 193.289,Z 193.064,A -85,B 0,C 180,E1 -24685.42,E2 -24685.42} C_VEL
LIN {X 0,Y 191.123,Z 205.964,A -85,B 0,C 180,E1 -24686.153,E2 -24686.153} C_VEL
LIN {X 0,Y 188.152,Z 218.219,A -85,B 0,C 180,E1 -24687.196,E2 -24687.196} C_VEL
LIN {X 0,Y 184.123,Z 230.402,A -85,B 0,C 180,E1 -24688.61,E2 -24688.61} C_VEL
LIN {X 0,Y 179.299,Z 242.037,A -85,B 0,C 180,E1 -24690.422,E2 -24690.422} C_VEL
LIN {X 0,Y 173.989,Z 252.351,A -85,B 0,C 180,E1 -24692.521,E2 -24692.521} C_VEL
LIN {X 0,Y 168.931,Z 260.773,A -85,B 0,C 180,E1 -24694.751,E2 -24694.751} C_VEL
LIN {X 0,Y 163.37,Z 268.811,A -85,B 0,C 180,E1 -24697.501,E2 -24697.501} C_VEL
LIN {X 0,Y 157.667,Z 275.994,A -85,B 0,C 180,E1 -24700.733,E2 -24700.733} C_VEL
LIN {X 0,Y 152.294,Z 282.003,A -85,B 0,C 180,E1 -24704.411,E2 -24704.411} C_VEL
LIN {X 0,Y 147.606,Z 286.528,A -85,B 0,C 180,E1 -24708.197,E2 -24708.197} C_VEL
LIN {X 0,Y 144.587,Z 289.064,A -85,B 0,C 180,E1 -24711.053,E2 -24711.053} C_VEL
LIN {X 0,Y 142.271,Z 290.854,A -85,B 0,C 180,E1 -24713.646,E2 -24713.646} C_VEL
LIN {X 0,Y 140.087,Z 292.325,A -85,B 0,C 180,E1 -24716.507,E2 -24716.507} C_VEL
LIN {X 0,Y 137.946,Z 293.469,A -85,B 0,C 180,E1 -24720.011,E2 -24720.011} C_VEL
LIN {X 0,Y 135.476,Z 294.104,A -85,B 0,C 180,E1 -24725.481,E2 -24725.481} C_VEL
LIN {X 0,Y 134.132,Z 293.455,A -85,B 0,C 180,E1 -24730.587,E2 -24730.587} C_VEL
LIN {X 0,Y 133.587,Z 292.084,A -85,B 0,C 180,E1 -24734.75,E2 -24734.75} C_VEL
LIN {X 0,Y 133.544,Z 290.579,A -85,B 0,C 180,E1 -24737.849,E2 -24737.849} C_VEL
LIN {X 0,Y 134.027,Z 287.482,A -85,B 0,C 180,E1 -24742.47,E2 -24742.47} C_VEL
LIN {X 0,Y 134.972,Z 283.335,A -85,B 0,C 180,E1 -24747.016,E2 -24747.016} C_VEL
LIN {X 0,Y 136.718,Z 277,A -85,B 0,C 180,E1 -24752.211,E2 -24752.211} C_VEL
LIN {X 0,Y 138.862,Z 270.121,A -85,B 0,C 180,E1 -24756.54,E2 -24756.54} C_VEL
LIN {X 0,Y 141.171,Z 263.096,A -85,B 0,C 180,E1 -24760.036,E2 -24760.036} C_VEL
LIN {X 0,Y 143.948,Z 254.626,A -85,B 0,C 180,E1 -24763.411,E2 -24763.411} C_VEL
LIN {X 0,Y 147.055,Z 244.175,A -85,B 0,C 180,E1 -24766.664,E2 -24766.664} C_VEL
LIN {X 0,Y 150.038,Z 232.443,A -85,B 0,C 180,E1 -24769.497,E2 -24769.497} C_VEL
LIN {X 0,Y 152.686,Z 220.653,A -85,B 0,C 180,E1 -24771.608,E2 -24771.608} C_VEL
LIN {X 0,Y 154.775,Z 208.451,A -85,B 0,C 180,E1 -24773.235,E2 -24773.235} C_VEL
LIN {X 0,Y 156.416,Z 195.227,A -85,B 0,C 180,E1 -24774.458,E2 -24774.458} C_VEL
LIN {X 0,Y 157.454,Z 180.853,A -85,B 0,C 180,E1 -24775.225,E2 -24775.225} C_VEL
LIN {X 0,Y 159.865,Z 138.431,A -85,B 0,C 180,E1 -24776.942,E2 -24776.942} C_VEL
LIN {X 0,Y 152.498,Z 122.767,A -85,B 0,C 180,E1 -24779.854,E2 -24779.854} C_VEL
LIN {X 0,Y 145.625,Z 110.742,A -85,B 0,C 180,E1 -24782.782,E2 -24782.782} C_VEL
LIN {X 0,Y 141.234,Z 104.054,A -85,B 0,C 180,E1 -24784.807,E2 -24784.807} C_VEL
LIN {X 0,Y 139.214,Z 100.842,A -85,B 0,C 180,E1 -24785.816,E2 -24785.816} C_VEL
LIN {X 0,Y 136.804,Z 97.946,A -85,B 0,C 180,E1 -24787.013,E2 -24787.013} C_VEL
LIN {X 0,Y 136.062,Z 95.537,A -85,B 0,C 180,E1 -24787.578,E2 -24787.578} C_VEL
LIN {X 0,Y 136.01,Z 95.536,A -85,B 0,C 180,E1 -24793.661,E2 -24793.661} C_VEL
LIN {X 0,Y 136.034,Z 95.538,A -85,B 0,C 180,E1 -24797.806,E2 -24797.806} C_VEL
LIN {X 0,Y 136.03,Z 95.498,A -85,B 0,C 180,E1 -24801.684,E2 -24801.684} C_VEL
LIN {X 0,Y 136.058,Z 95.479,A -85,B 0,C 180,E1 -24805.74,E2 -24805.74} C_VEL
LIN {X 0,Y 136.15,Z 95.525,A -85,B 0,C 180,E1 -24812.316,E2 -24812.316} C_VEL
LIN {X 0,Y 136.247,Z 95.512,A -85,B 0,C 180,E1 -24818.833,E2 -24818.833} C_VEL
LIN {X 0,Y 136.272,Z 95.496,A -85,B 0,C 180,E1 -24825.056,E2 -24825.056} C_VEL
LIN {X 0,Y 136.448,Z 95.488,A -85,B 0,C 180,E1 -24828.137,E2 -24828.137} C_VEL
LIN {X 0,Y 136.555,Z 95.458,A -85,B 0,C 180,E1 -24831.117,E2 -24831.117} C_VEL
LIN {X 0,Y 137.136,Z 95.385,A -85,B 0,C 180,E1 -24839.999,E2 -24839.999} C_VEL
LIN {X 0,Y 136.553,Z 95.46,A -85,B 0,C 180,E1 -24848.881,E2 -24848.881} C_VEL
LIN {X 0,Y 136.443,Z 95.489,A -85,B 0,C 180,E1 -24851.889,E2 -24851.889} C_VEL
LIN {X 0,Y 136.24,Z 95.512,A -85,B 0,C 180,E1 -24858.029,E2 -24858.029} C_VEL
LIN {X 0,Y 136.199,Z 95.515,A -85,B 0,C 180,E1 -24861.746,E2 -24861.746} C_VEL
LIN {X 0,Y 136.101,Z 95.523,A -85,B 0,C 180,E1 -24868.614,E2 -24868.614} C_VEL
LIN {X 0,Y 136.073,Z 95.533,A -85,B 0,C 180,E1 -24874.62,E2 -24874.62} C_VEL
LIN {X 0,Y 136.04,Z 95.546,A -85,B 0,C 180,E1 -24877.724,E2 -24877.724} C_VEL
LIN {X 0,Y 136.964,Z 98.245,A -85,B 0,C 180,E1 -24878.315,E2 -24878.315} C_VEL
LIN {X 0,Y 139.223,Z 101.003,A -85,B 0,C 180,E1 -24879.432,E2 -24879.432} C_VEL
LIN {X 0,Y 141.294,Z 104.202,A -85,B 0,C 180,E1 -24880.456,E2 -24880.456} C_VEL
LIN {X 0,Y 143.214,Z 107.524,A -85,B 0,C 180,E1 -24881.39,E2 -24881.39} C_VEL
LIN {X 0,Y 148.458,Z 118.05,A -85,B 0,C 180,E1 -24883.856,E2 -24883.856} C_VEL
LIN {X 0,Y 153.003,Z 128.796,A -85,B 0,C 180,E1 -24885.889,E2 -24885.889} C_VEL
LIN {X 0,Y 156.772,Z 139.597,A -85,B 0,C 180,E1 -24887.553,E2 -24887.553} C_VEL
LIN {X 0,Y 158.544,Z 164.538,A -85,B 0,C 180,E1 -24889.386,E2 -24889.386} C_VEL
LIN {X 0,Y 156.228,Z 204.347,A -85,B 0,C 180,E1 -24891.067,E2 -24891.067} C_VEL
LIN {X 0,Y 154.731,Z 217.648,A -85,B 0,C 180,E1 -24892.076,E2 -24892.076} C_VEL
LIN {X 0,Y 152.845,Z 228.683,A -85,B 0,C 180,E1 -24893.29,E2 -24893.29} C_VEL
LIN {X 0,Y 150.299,Z 240.425,A -85,B 0,C 180,E1 -24895.052,E2 -24895.052} C_VEL
LIN {X 0,Y 147.11,Z 252.42,A -85,B 0,C 180,E1 -24897.488,E2 -24897.488} C_VEL
LIN {X 0,Y 144.352,Z 262.061,A -85,B 0,C 180,E1 -24900.063,E2 -24900.063} C_VEL
LIN {X 0,Y 141.308,Z 271.895,A -85,B 0,C 180,E1 -24903.408,E2 -24903.408} C_VEL
LIN {X 0,Y 139.164,Z 278.425,A -85,B 0,C 180,E1 -24906.17,E2 -24906.17} C_VEL
LIN {X 0,Y 136.785,Z 286.611,A -85,B 0,C 180,E1 -24910.489,E2 -24910.489} C_VEL
LIN {X 0,Y 134.993,Z 293.147,A -85,B 0,C 180,E1 -24914.91,E2 -24914.91} C_VEL
LIN {X 0,Y 134.057,Z 298.325,A -85,B 0,C 180,E1 -24919.426,E2 -24919.426} C_VEL
LIN {X 0,Y 133.838,Z 302.324,A -85,B 0,C 180,E1 -24923.97,E2 -24923.97} C_VEL
LIN {X 0,Y 133.847,Z 304.354,A -85,B 0,C 180,E1 -24926.989,E2 -24926.989} C_VEL
LIN {X 0,Y 134.046,Z 305.954,A -85,B 0,C 180,E1 -24929.999,E2 -24929.999} C_VEL
LIN {X 0,Y 133.808,Z 307.28,A -85,B 0,C 180,E1 -24933.687,E2 -24933.687} C_VEL
LIN {X 0,Y 133.846,Z 308.093,A -85,B 0,C 180,E1 -24939.062,E2 -24939.062} C_VEL
LIN {X 0,Y 135.168,Z 307.567,A -85,B 0,C 180,E1 -24945.067,E2 -24945.067} C_VEL
LIN {X 0,Y 136.837,Z 306.317,A -85,B 0,C 180,E1 -24948.966,E2 -24948.966} C_VEL
LIN {X 0,Y 137.611,Z 305.26,A -85,B 0,C 180,E1 -24951.371,E2 -24951.371} C_VEL
LIN {X 0,Y 137.601,Z 302.986,A -85,B 0,C 180,E1 -24955.401,E2 -24955.401} C_VEL
LIN {X 0,Y 137.899,Z 300.745,A -85,B 0,C 180,E1 -24958.579,E2 -24958.579} C_VEL
LIN {X 0,Y 139.124,Z 298.764,A -85,B 0,C 180,E1 -24960.831,E2 -24960.831} C_VEL
LIN {X 0,Y 139.822,Z 298.016,A -85,B 0,C 180,E1 -24961.529,E2 -24961.529} C_VEL
LIN {X 0,Y 145.074,Z 292.786,A -85,B 0,C 180,E1 -24965.543,E2 -24965.543} C_VEL
LIN {X 0,Y 150.758,Z 286.593,A -85,B 0,C 180,E1 -24969,E2 -24969} C_VEL
LIN {X 0,Y 157.004,Z 278.93,A -85,B 0,C 180,E1 -24972.178,E2 -24972.178} C_VEL
LIN {X 0,Y 162.557,Z 271.125,A -85,B 0,C 180,E1 -24974.631,E2 -24974.631} C_VEL
LIN {X 0,Y 167.848,Z 262.692,A -85,B 0,C 180,E1 -24976.677,E2 -24976.677} C_VEL
LIN {X 0,Y 173.446,Z 252.401,A -85,B 0,C 180,E1 -24978.556,E2 -24978.556} C_VEL
LIN {X 0,Y 178.639,Z 241.006,A -85,B 0,C 180,E1 -24980.099,E2 -24980.099} C_VEL
LIN {X 0,Y 183.103,Z 228.626,A -85,B 0,C 180,E1 -24981.335,E2 -24981.335} C_VEL
LIN {X 0,Y 186.555,Z 215.373,A -85,B 0,C 180,E1 -24982.289,E2 -24982.289} C_VEL
LIN {X 0,Y 188.832,Z 202.567,A -85,B 0,C 180,E1 -24982.889,E2 -24982.889} C_VEL
LIN {X 0,Y 190.614,Z 182.429,A -85,B 0,C 180,E1 -24983.564,E2 -24983.564} C_VEL
LIN {X 0,Y 187.75,Z 174.392,A -85,B 0,C 180,E1 -24985.72,E2 -24985.72} C_VEL
LIN {X 0,Y 183.988,Z 165.265,A -85,B 0,C 180,E1 -24988.81,E2 -24988.81} C_VEL
LIN {X 0,Y 180.82,Z 158.268,A -85,B 0,C 180,E1 -24991.765,E2 -24991.765} C_VEL
LIN {X 0,Y 178.597,Z 153.76,A -85,B 0,C 180,E1 -24994.112,E2 -24994.112} C_VEL
LIN {X 0,Y 176.465,Z 149.429,A -85,B 0,C 180,E1 -24996.714,E2 -24996.714} C_VEL
LIN {X 0,Y 174.148,Z 144.955,A -85,B 0,C 180,E1 -25000.171,E2 -25000.171} C_VEL
LIN {X 0,Y 172.432,Z 142.336,A -85,B 0,C 180,E1 -25003.423,E2 -25003.423} C_VEL
LIN {X 0,Y 171.125,Z 139.172,A -85,B 0,C 180,E1 -25007.392,E2 -25007.392} C_VEL
LIN {X 0,Y 170.213,Z 138.625,A -85,B 0,C 180,E1 -25012.885,E2 -25012.885} C_VEL
LIN {X 0,Y 171.212,Z 138.923,A -85,B 0,C 180,E1 -25019.564,E2 -25019.564} C_VEL
LIN {X 0,Y 172.756,Z 142.44,A -85,B 0,C 180,E1 -25023.961,E2 -25023.961} C_VEL
LIN {X 0,Y 174.238,Z 144.158,A -85,B 0,C 180,E1 -25026.587,E2 -25026.587} C_VEL
LIN {X 0,Y 176.544,Z 147.928,A -85,B 0,C 180,E1 -25029.952,E2 -25029.952} C_VEL
LIN {X 0,Y 177.593,Z 149.523,A -85,B 0,C 180,E1 -25031.222,E2 -25031.222} C_VEL
LIN {X 0,Y 179.96,Z 153.267,A -85,B 0,C 180,E1 -25033.788,E2 -25033.788} C_VEL
LIN {X 0,Y 182.857,Z 158.012,A -85,B 0,C 180,E1 -25036.508,E2 -25036.508} C_VEL
LIN {X 0,Y 187.03,Z 165.251,A -85,B 0,C 180,E1 -25039.887,E2 -25039.887} C_VEL
LIN {X 0,Y 191.35,Z 173.674,A -85,B 0,C 180,E1 -25042.95,E2 -25042.95} C_VEL
LIN {X 0,Y 189.44,Z 193.894,A -85,B 0,C 180,E1 -25043.65,E2 -25043.65} C_VEL
LIN {X 0,Y 187.103,Z 207.1,A -85,B 0,C 180,E1 -25044.406,E2 -25044.406} C_VEL
LIN {X 0,Y 183.917,Z 219.437,A -85,B 0,C 180,E1 -25045.476,E2 -25045.476} C_VEL
LIN {X 0,Y 180.068,Z 230.63,A -85,B 0,C 180,E1 -25046.775,E2 -25046.775} C_VEL
LIN {X 0,Y 175.009,Z 242.404,A -85,B 0,C 180,E1 -25048.595,E2 -25048.595} C_VEL
LIN {X 0,Y 169.534,Z 252.64,A -85,B 0,C 180,E1 -25050.665,E2 -25050.665} C_VEL
LIN {X 0,Y 163.699,Z 261.917,A -85,B 0,C 180,E1 -25053.158,E2 -25053.158} C_VEL
LIN {X 0,Y 157.858,Z 269.871,A -85,B 0,C 180,E1 -25055.948,E2 -25055.948} C_VEL
LIN {X 0,Y 151.939,Z 276.893,A -85,B 0,C 180,E1 -25059.217,E2 -25059.217} C_VEL
LIN {X 0,Y 146.887,Z 282.206,A -85,B 0,C 180,E1 -25062.558,E2 -25062.558} C_VEL
LIN {X 0,Y 142.16,Z 286.547,A -85,B 0,C 180,E1 -25066.203,E2 -25066.203} C_VEL
LIN {X 0,Y 138.393,Z 289.533,A -85,B 0,C 180,E1 -25069.62,E2 -25069.62} C_VEL
LIN {X 0,Y 133.961,Z 292.542,A -85,B 0,C 180,E1 -25074.755,E2 -25074.755} C_VEL
LIN {X 0,Y 131.234,Z 293.894,A -85,B 0,C 180,E1 -25078.967,E2 -25078.967} C_VEL
LIN {X 0,Y 128.796,Z 294.482,A -85,B 0,C 180,E1 -25084.118,E2 -25084.118} C_VEL
LIN {X 0,Y 127.126,Z 293.825,A -85,B 0,C 180,E1 -25090.025,E2 -25090.025} C_VEL
LIN {X 0,Y 126.569,Z 292.64,A -85,B 0,C 180,E1 -25093.882,E2 -25093.882} C_VEL
LIN {X 0,Y 126.426,Z 291.211,A -85,B 0,C 180,E1 -25097.154,E2 -25097.154} C_VEL
LIN {X 0,Y 126.849,Z 288.203,A -85,B 0,C 180,E1 -25102.039,E2 -25102.039} C_VEL
LIN {X 0,Y 127.811,Z 284.156,A -85,B 0,C 180,E1 -25106.849,E2 -25106.849} C_VEL
LIN {X 0,Y 129.553,Z 277.959,A -85,B 0,C 180,E1 -25112.333,E2 -25112.333} C_VEL
LIN {X 0,Y 131.772,Z 271.202,A -85,B 0,C 180,E1 -25116.893,E2 -25116.893} C_VEL
LIN {X 0,Y 134.702,Z 262.815,A -85,B 0,C 180,E1 -25121.284,E2 -25121.284} C_VEL
LIN {X 0,Y 137.666,Z 254.163,A -85,B 0,C 180,E1 -25124.79,E2 -25124.79} C_VEL
LIN {X 0,Y 140.96,Z 243.523,A -85,B 0,C 180,E1 -25128.158,E2 -25128.158} C_VEL
LIN {X 0,Y 143.745,Z 233.002,A -85,B 0,C 180,E1 -25130.762,E2 -25130.762} C_VEL
LIN {X 0,Y 146.505,Z 221.287,A -85,B 0,C 180,E1 -25132.941,E2 -25132.941} C_VEL
LIN {X 0,Y 148.719,Z 209.151,A -85,B 0,C 180,E1 -25134.612,E2 -25134.612} C_VEL
LIN {X 0,Y 150.423,Z 196.194,A -85,B 0,C 180,E1 -25135.86,E2 -25135.86} C_VEL
LIN {X 0,Y 151.476,Z 182.659,A -85,B 0,C 180,E1 -25136.638,E2 -25136.638} C_VEL
LIN {X 0,Y 154.001,Z 140.489,A -85,B 0,C 180,E1 -25138.384,E2 -25138.384} C_VEL
LIN {X 0,Y 147.082,Z 125.654,A -85,B 0,C 180,E1 -25141.345,E2 -25141.345} C_VEL
LIN {X 0,Y 139.78,Z 113.002,A -85,B 0,C 180,E1 -25144.738,E2 -25144.738} C_VEL
LIN {X 0,Y 134.79,Z 105.535,A -85,B 0,C 180,E1 -25147.304,E2 -25147.304} C_VEL
LIN {X 0,Y 132.564,Z 102.353,A -85,B 0,C 180,E1 -25148.534,E2 -25148.534} C_VEL
LIN {X 0,Y 131.845,Z 101.246,A -85,B 0,C 180,E1 -25148.953,E2 -25148.953} C_VEL
LIN {X 0,Y 129.812,Z 98.961,A -85,B 0,C 180,E1 -25150.111,E2 -25150.111} C_VEL
LIN {X 0,Y 128.957,Z 96.414,A -85,B 0,C 180,E1 -25150.844,E2 -25150.844} C_VEL
LIN {X 0,Y 128.929,Z 96.412,A -85,B 0,C 180,E1 -25155.126,E2 -25155.126} C_VEL
LIN {X 0,Y 128.951,Z 96.408,A -85,B 0,C 180,E1 -25159.732,E2 -25159.732} C_VEL
LIN {X 0,Y 128.961,Z 96.357,A -85,B 0,C 180,E1 -25164.833,E2 -25164.833} C_VEL
LIN {X 0,Y 129.055,Z 96.406,A -85,B 0,C 180,E1 -25170.651,E2 -25170.651} C_VEL
LIN {X 0,Y 129.111,Z 96.394,A -85,B 0,C 180,E1 -25177.727,E2 -25177.727} C_VEL
LIN {X 0,Y 129.157,Z 96.393,A -85,B 0,C 180,E1 -25180.943,E2 -25180.943} C_VEL
LIN {X 0,Y 129.37,Z 96.37,A -85,B 0,C 180,E1 -25187.922,E2 -25187.922} C_VEL
LIN {X 0,Y 129.48,Z 96.342,A -85,B 0,C 180,E1 -25190.628,E2 -25190.628} C_VEL
LIN {X 0,Y 130.091,Z 96.262,A -85,B 0,C 180,E1 -25199.999,E2 -25199.999} C_VEL
LIN {X 0,Y 129.476,Z 96.344,A -85,B 0,C 180,E1 -25209.371,E2 -25209.371} C_VEL
LIN {X 0,Y 129.346,Z 96.373,A -85,B 0,C 180,E1 -25212.552,E2 -25212.552} C_VEL
LIN {X 0,Y 129.153,Z 96.398,A -85,B 0,C 180,E1 -25219.056,E2 -25219.056} C_VEL
LIN {X 0,Y 129.11,Z 96.4,A -85,B 0,C 180,E1 -25222.397,E2 -25222.397} C_VEL
LIN {X 0,Y 129.029,Z 96.407,A -85,B 0,C 180,E1 -25225.832,E2 -25225.832} C_VEL
LIN {X 0,Y 129.018,Z 96.399,A -85,B 0,C 180,E1 -25229.357,E2 -25229.357} C_VEL
LIN {X 0,Y 129.065,Z 96.52,A -85,B 0,C 180,E1 -25234.552,E2 -25234.552} C_VEL
LIN {X 0,Y 129.959,Z 99.183,A -85,B 0,C 180,E1 -25235.218,E2 -25235.218} C_VEL
LIN {X 0,Y 132.341,Z 101.899,A -85,B 0,C 180,E1 -25236.567,E2 -25236.567} C_VEL
LIN {X 0,Y 134.321,Z 105.083,A -85,B 0,C 180,E1 -25237.699,E2 -25237.699} C_VEL
LIN {X 0,Y 135.865,Z 107.247,A -85,B 0,C 180,E1 -25238.519,E2 -25238.519} C_VEL
LIN {X 0,Y 138.311,Z 111.116,A -85,B 0,C 180,E1 -25239.791,E2 -25239.791} C_VEL
LIN {X 0,Y 142.683,Z 119.903,A -85,B 0,C 180,E1 -25242.029,E2 -25242.029} C_VEL
LIN {X 0,Y 147.086,Z 130.11,A -85,B 0,C 180,E1 -25244.17,E2 -25244.17} C_VEL
LIN {X 0,Y 151.177,Z 141.923,A -85,B 0,C 180,E1 -25246.136,E2 -25246.136} C_VEL
LIN {X 0,Y 152.707,Z 165.99,A -85,B 0,C 180,E1 -25247.966,E2 -25247.966} C_VEL
LIN {X 0,Y 150.257,Z 204.684,A -85,B 0,C 180,E1 -25249.644,E2 -25249.644} C_VEL
LIN {X 0,Y 148.571,Z 218.514,A -85,B 0,C 180,E1 -25250.75,E2 -25250.75} C_VEL
LIN {X 0,Y 146.52,Z 229.806,A -85,B 0,C 180,E1 -25252.079,E2 -25252.079} C_VEL
LIN {X 0,Y 143.684,Z 241.98,A -85,B 0,C 180,E1 -25254.058,E2 -25254.058} C_VEL
LIN {X 0,Y 140.337,Z 253.547,A -85,B 0,C 180,E1 -25256.572,E2 -25256.572} C_VEL
LIN {X 0,Y 137.457,Z 262.924,A -85,B 0,C 180,E1 -25259.249,E2 -25259.249} C_VEL
LIN {X 0,Y 134.555,Z 271.933,A -85,B 0,C 180,E1 -25262.512,E2 -25262.512} C_VEL
LIN {X 0,Y 132.586,Z 277.397,A -85,B 0,C 180,E1 -25264.908,E2 -25264.908} C_VEL
LIN {X 0,Y 130.416,Z 284.444,A -85,B 0,C 180,E1 -25268.668,E2 -25268.668} C_VEL
LIN {X 0,Y 128.367,Z 291.319,A -85,B 0,C 180,E1 -25273.295,E2 -25273.295} C_VEL
LIN {X 0,Y 127.029,Z 297.622,A -85,B 0,C 180,E1 -25278.834,E2 -25278.834} C_VEL
LIN {X 0,Y 126.739,Z 301.701,A -85,B 0,C 180,E1 -25283.631,E2 -25283.631} C_VEL
LIN {X 0,Y 126.787,Z 303.784,A -85,B 0,C 180,E1 -25286.821,E2 -25286.821} C_VEL
LIN {X 0,Y 126.963,Z 305.417,A -85,B 0,C 180,E1 -25289.999,E2 -25289.999} C_VEL
LIN {X 0,Y 126.739,Z 306.699,A -85,B 0,C 180,E1 -25293.5,E2 -25293.5} C_VEL
LIN {X 0,Y 126.829,Z 307.69,A -85,B 0,C 180,E1 -25299.568,E2 -25299.568} C_VEL
LIN {X 0,Y 128.296,Z 307.23,A -85,B 0,C 180,E1 -25305.895,E2 -25305.895} C_VEL
LIN {X 0,Y 129.938,Z 306.172,A -85,B 0,C 180,E1 -25309.667,E2 -25309.667} C_VEL
LIN {X 0,Y 133.441,Z 303.624,A -85,B 0,C 180,E1 -25314.918,E2 -25314.918} C_VEL
LIN {X 0,Y 137.884,Z 299.836,A -85,B 0,C 180,E1 -25319.755,E2 -25319.755} C_VEL
LIN {X 0,Y 139.822,Z 298.016,A -85,B 0,C 180,E1 -25321.529,E2 -25321.529} C_VEL
LIN {X 0,Y 141.649,Z 295.726,A -85,B 0,C 180,E1 -25323.622,E2 -25323.622} C_VEL
LIN {X 0,Y 143.44,Z 291.601,A -85,B 0,C 180,E1 -25327.179,E2 -25327.179} C_VEL
LIN {X 0,Y 145.661,Z 286.873,A -85,B 0,C 180,E1 -25330.508,E2 -25330.508} C_VEL
LIN {X 0,Y 148.066,Z 283.622,A -85,B 0,C 180,E1 -25332.181,E2 -25332.181} C_VEL
LIN {X 0,Y 154.067,Z 276.222,A -85,B 0,C 180,E1 -25334.994,E2 -25334.994} C_VEL
LIN {X 0,Y 157.604,Z 271.466,A -85,B 0,C 180,E1 -25336.437,E2 -25336.437} C_VEL
LIN {X 0,Y 162.42,Z 264.158,A -85,B 0,C 180,E1 -25338.28,E2 -25338.28} C_VEL
LIN {X 0,Y 168.182,Z 254.351,A -85,B 0,C 180,E1 -25340.16,E2 -25340.16} C_VEL
LIN {X 0,Y 173.496,Z 243.568,A -85,B 0,C 180,E1 -25341.705,E2 -25341.705} C_VEL
LIN {X 0,Y 178.242,Z 231.636,A -85,B 0,C 180,E1 -25342.948,E2 -25342.948} C_VEL
LIN {X 0,Y 181.965,Z 219.272,A -85,B 0,C 180,E1 -25343.907,E2 -25343.907} C_VEL
LIN {X 0,Y 184.677,Z 206.376,A -85,B 0,C 180,E1 -25344.598,E2 -25344.598} C_VEL
LIN {X 0,Y 186.477,Z 190.59,A -85,B 0,C 180,E1 -25345.143,E2 -25345.143} C_VEL
LIN {X 0,Y 186.868,Z 185.091,A -85,B 0,C 180,E1 -25345.362,E2 -25345.362} C_VEL
LIN {X 0,Y 183.689,Z 176.206,A -85,B 0,C 180,E1 -25348.019,E2 -25348.019} C_VEL
LIN {X 0,Y 180.336,Z 167.916,A -85,B 0,C 180,E1 -25351.138,E2 -25351.138} C_VEL
LIN {X 0,Y 177.508,Z 161.386,A -85,B 0,C 180,E1 -25354.182,E2 -25354.182} C_VEL
LIN {X 0,Y 174.727,Z 155.664,A -85,B 0,C 180,E1 -25357.721,E2 -25357.721} C_VEL
LIN {X 0,Y 172.73,Z 151.496,A -85,B 0,C 180,E1 -25361.004,E2 -25361.004} C_VEL
LIN {X 0,Y 170.149,Z 146.182,A -85,B 0,C 180,E1 -25367.701,E2 -25367.701} C_VEL
LIN {X 0,Y 169.376,Z 145.69,A -85,B 0,C 180,E1 -25374.764,E2 -25374.764} C_VEL
LIN {X 0,Y 170.248,Z 146.03,A -85,B 0,C 180,E1 -25379.342,E2 -25379.342} C_VEL
LIN {X 0,Y 171.692,Z 149.364,A -85,B 0,C 180,E1 -25383.63,E2 -25383.63} C_VEL
LIN {X 0,Y 172.951,Z 150.967,A -85,B 0,C 180,E1 -25385.996,E2 -25385.996} C_VEL
LIN {X 0,Y 175.33,Z 154.886,A -85,B 0,C 180,E1 -25389.624,E2 -25389.624} C_VEL
LIN {X 0,Y 178.341,Z 159.952,A -85,B 0,C 180,E1 -25393.17,E2 -25393.17} C_VEL
LIN {X 0,Y 181.703,Z 165.693,A -85,B 0,C 180,E1 -25396.43,E2 -25396.43} C_VEL
LIN {X 0,Y 185.878,Z 173.585,A -85,B 0,C 180,E1 -25399.895,E2 -25399.895} C_VEL
LIN {X 0,Y 187.585,Z 177.251,A -85,B 0,C 180,E1 -25401.194,E2 -25401.194} C_VEL
LIN {X 0,Y 185.831,Z 194.51,A -85,B 0,C 180,E1 -25401.794,E2 -25401.794} C_VEL
LIN {X 0,Y 183.46,Z 207.409,A -85,B 0,C 180,E1 -25402.525,E2 -25402.525} C_VEL
LIN {X 0,Y 180.195,Z 219.669,A -85,B 0,C 180,E1 -25403.575,E2 -25403.575} C_VEL
LIN {X 0,Y 176.209,Z 230.884,A -85,B 0,C 180,E1 -25404.858,E2 -25404.858} C_VEL
LIN {X 0,Y 171.423,Z 241.69,A -85,B 0,C 180,E1 -25406.488,E2 -25406.488} C_VEL
LIN {X 0,Y 165.902,Z 251.902,A -85,B 0,C 180,E1 -25408.478,E2 -25408.478} C_VEL
LIN {X 0,Y 159.779,Z 261.385,A -85,B 0,C 180,E1 -25410.94,E2 -25410.94} C_VEL
LIN {X 0,Y 153.799,Z 269.299,A -85,B 0,C 180,E1 -25413.641,E2 -25413.641} C_VEL
LIN {X 0,Y 147.347,Z 276.654,A -85,B 0,C 180,E1 -25416.975,E2 -25416.975} C_VEL
LIN {X 0,Y 141.661,Z 282.392,A -85,B 0,C 180,E1 -25420.562,E2 -25420.562} C_VEL
LIN {X 0,Y 136.891,Z 286.539,A -85,B 0,C 180,E1 -25424.049,E2 -25424.049} C_VEL
LIN {X 0,Y 132.333,Z 289.984,A -85,B 0,C 180,E1 -25428.033,E2 -25428.033} C_VEL
LIN {X 0,Y 127.978,Z 292.734,A -85,B 0,C 180,E1 -25432.839,E2 -25432.839} C_VEL
LIN {X 0,Y 124.621,Z 294.31,A -85,B 0,C 180,E1 -25437.773,E2 -25437.773} C_VEL
LIN {X 0,Y 122.193,Z 294.858,A -85,B 0,C 180,E1 -25442.606,E2 -25442.606} C_VEL
LIN {X 0,Y 121.001,Z 294.737,A -85,B 0,C 180,E1 -25446.012,E2 -25446.012} C_VEL
LIN {X 0,Y 120.133,Z 294.178,A -85,B 0,C 180,E1 -25449.452,E2 -25449.452} C_VEL
LIN {X 0,Y 119.571,Z 293.194,A -85,B 0,C 180,E1 -25452.911,E2 -25452.911} C_VEL
LIN {X 0,Y 119.328,Z 291.811,A -85,B 0,C 180,E1 -25456.375,E2 -25456.375} C_VEL
LIN {X 0,Y 119.686,Z 288.895,A -85,B 0,C 180,E1 -25461.56,E2 -25461.56} C_VEL
LIN {X 0,Y 120.65,Z 284.944,A -85,B 0,C 180,E1 -25466.662,E2 -25466.662} C_VEL
LIN {X 0,Y 122.123,Z 279.873,A -85,B 0,C 180,E1 -25471.65,E2 -25471.65} C_VEL
LIN {X 0,Y 124.292,Z 273.508,A -85,B 0,C 180,E1 -25476.495,E2 -25476.495} C_VEL
LIN {X 0,Y 127.17,Z 265.533,A -85,B 0,C 180,E1 -25481.154,E2 -25481.154} C_VEL
LIN {X 0,Y 130.122,Z 257.402,A -85,B 0,C 180,E1 -25484.867,E2 -25484.867} C_VEL
LIN {X 0,Y 133.518,Z 247.486,A -85,B 0,C 180,E1 -25488.412,E2 -25488.412} C_VEL
LIN {X 0,Y 136.783,Z 236.383,A -85,B 0,C 180,E1 -25491.476,E2 -25491.476} C_VEL
LIN {X 0,Y 139.535,Z 225.511,A -85,B 0,C 180,E1 -25493.763,E2 -25493.763} C_VEL
LIN {X 0,Y 142.107,Z 213.49,A -85,B 0,C 180,E1 -25495.642,E2 -25495.642} C_VEL
LIN {X 0,Y 144.083,Z 200.952,A -85,B 0,C 180,E1 -25497.047,E2 -25497.047} C_VEL
LIN {X 0,Y 145.404,Z 187.547,A -85,B 0,C 180,E1 -25497.998,E2 -25497.998} C_VEL
LIN {X 0,Y 148.223,Z 142.551,A -85,B 0,C 180,E1 -25499.939,E2 -25499.939} C_VEL
LIN {X 0,Y 141.996,Z 129.181,A -85,B 0,C 180,E1 -25502.826,E2 -25502.826} C_VEL
LIN {X 0,Y 135.628,Z 117.835,A -85,B 0,C 180,E1 -25506.037,E2 -25506.037} C_VEL
LIN {X 0,Y 130.617,Z 110.345,A -85,B 0,C 180,E1 -25508.801,E2 -25508.801} C_VEL
LIN {X 0,Y 127.921,Z 106.437,A -85,B 0,C 180,E1 -25510.432,E2 -25510.432} C_VEL
LIN {X 0,Y 125.845,Z 103.582,A -85,B 0,C 180,E1 -25511.76,E2 -25511.76} C_VEL
LIN {X 0,Y 125.162,Z 102.455,A -85,B 0,C 180,E1 -25512.231,E2 -25512.231} C_VEL
LIN {X 0,Y 123.116,Z 100.554,A -85,B 0,C 180,E1 -25513.564,E2 -25513.564} C_VEL
LIN {X 0,Y 122.035,Z 98.127,A -85,B 0,C 180,E1 -25514.438,E2 -25514.438} C_VEL
LIN {X 0,Y 121.865,Z 97.292,A -85,B 0,C 180,E1 -25514.624,E2 -25514.624} C_VEL
LIN {X 0,Y 121.865,Z 97.272,A -85,B 0,C 180,E1 -25520.625,E2 -25520.625} C_VEL
LIN {X 0,Y 121.913,Z 97.233,A -85,B 0,C 180,E1 -25524.796,E2 -25524.796} C_VEL
LIN {X 0,Y 121.943,Z 97.285,A -85,B 0,C 180,E1 -25529.828,E2 -25529.828} C_VEL
LIN {X 0,Y 121.987,Z 97.271,A -85,B 0,C 180,E1 -25536.215,E2 -25536.215} C_VEL
LIN {X 0,Y 122.05,Z 97.282,A -85,B 0,C 180,E1 -25539.787,E2 -25539.787} C_VEL
LIN {X 0,Y 122.243,Z 97.254,A -85,B 0,C 180,E1 -25546.704,E2 -25546.704} C_VEL
LIN {X 0,Y 122.41,Z 97.226,A -85,B 0,C 180,E1 -25550.081,E2 -25550.081} C_VEL
LIN {X 0,Y 122.602,Z 97.211,A -85,B 0,C 180,E1 -25556.713,E2 -25556.713} C_VEL
LIN {X 0,Y 123.045,Z 97.139,A -85,B 0,C 180,E1 -25559.999,E2 -25559.999} C_VEL
LIN {X 0,Y 122.426,Z 97.223,A -85,B 0,C 180,E1 -25566.592,E2 -25566.592} C_VEL
LIN {X 0,Y 122.325,Z 97.248,A -85,B 0,C 180,E1 -25572.385,E2 -25572.385} C_VEL
LIN {X 0,Y 122.107,Z 97.262,A -85,B 0,C 180,E1 -25576.724,E2 -25576.724} C_VEL
LIN {X 0,Y 122.03,Z 97.283,A -85,B 0,C 180,E1 -25582.854,E2 -25582.854} C_VEL
LIN {X 0,Y 121.942,Z 97.293,A -85,B 0,C 180,E1 -25587.456,E2 -25587.456} C_VEL
LIN {X 0,Y 121.927,Z 97.279,A -85,B 0,C 180,E1 -25590.579,E2 -25590.579} C_VEL
LIN {X 0,Y 122.856,Z 100.03,A -85,B 0,C 180,E1 -25591.466,E2 -25591.466} C_VEL
LIN {X 0,Y 124.847,Z 102.186,A -85,B 0,C 180,E1 -25592.807,E2 -25592.807} C_VEL
LIN {X 0,Y 125.611,Z 102.996,A -85,B 0,C 180,E1 -25593.299,E2 -25593.299} C_VEL
LIN {X 0,Y 127.609,Z 106.157,A -85,B 0,C 180,E1 -25594.624,E2 -25594.624} C_VEL
LIN {X 0,Y 128.93,Z 107.841,A -85,B 0,C 180,E1 -25595.425,E2 -25595.425} C_VEL
LIN {X 0,Y 133.727,Z 115.033,A -85,B 0,C 180,E1 -25598.194,E2 -25598.194} C_VEL
LIN {X 0,Y 138.791,Z 125.566,A -85,B 0,C 180,E1 -25600.993,E2 -25600.993} C_VEL
LIN {X 0,Y 143.206,Z 136.66,A -85,B 0,C 180,E1 -25603.314,E2 -25603.314} C_VEL
LIN {X 0,Y 145.666,Z 144.243,A -85,B 0,C 180,E1 -25604.605,E2 -25604.605} C_VEL
LIN {X 0,Y 146.951,Z 166.333,A -85,B 0,C 180,E1 -25606.365,E2 -25606.365} C_VEL
LIN {X 0,Y 144.509,Z 203.863,A -85,B 0,C 180,E1 -25608.031,E2 -25608.031} C_VEL
LIN {X 0,Y 142.75,Z 217.846,A -85,B 0,C 180,E1 -25609.164,E2 -25609.164} C_VEL
LIN {X 0,Y 140.471,Z 229.774,A -85,B 0,C 180,E1 -25610.595,E2 -25610.595} C_VEL
LIN {X 0,Y 137.523,Z 241.851,A -85,B 0,C 180,E1 -25612.636,E2 -25612.636} C_VEL
LIN {X 0,Y 134.017,Z 253.37,A -85,B 0,C 180,E1 -25615.228,E2 -25615.228} C_VEL
LIN {X 0,Y 130.997,Z 262.713,A -85,B 0,C 180,E1 -25618.007,E2 -25618.007} C_VEL
LIN {X 0,Y 128.143,Z 271.177,A -85,B 0,C 180,E1 -25621.2,E2 -25621.2} C_VEL
LIN {X 0,Y 125.623,Z 277.892,A -85,B 0,C 180,E1 -25624.304,E2 -25624.304} C_VEL
LIN {X 0,Y 122.973,Z 286.041,A -85,B 0,C 180,E1 -25629.071,E2 -25629.071} C_VEL
LIN {X 0,Y 121.231,Z 291.526,A -85,B 0,C 180,E1 -25633.149,E2 -25633.149} C_VEL
LIN {X 0,Y 120.034,Z 296.896,A -85,B 0,C 180,E1 -25638.174,E2 -25638.174} C_VEL
LIN {X 0,Y 119.655,Z 301.055,A -85,B 0,C 180,E1 -25643.253,E2 -25643.253} C_VEL
LIN {X 0,Y 119.722,Z 303.212,A -85,B 0,C 180,E1 -25646.633,E2 -25646.633} C_VEL
LIN {X 0,Y 119.883,Z 304.88,A -85,B 0,C 180,E1 -25649.999,E2 -25649.999} C_VEL
LIN {X 0,Y 119.681,Z 306.09,A -85,B 0,C 180,E1 -25653.365,E2 -25653.365} C_VEL
LIN {X 0,Y 119.551,Z 306.892,A -85,B 0,C 180,E1 -25656.751,E2 -25656.751} C_VEL
LIN {X 0,Y 119.806,Z 307.286,A -85,B 0,C 180,E1 -25660.135,E2 -25660.135} C_VEL
LIN {X 0,Y 121.436,Z 306.893,A -85,B 0,C 180,E1 -25666.819,E2 -25666.819} C_VEL
LIN {X 0,Y 124.788,Z 305.004,A -85,B 0,C 180,E1 -25673.217,E2 -25673.217} C_VEL
LIN {X 0,Y 127.02,Z 303.432,A -85,B 0,C 180,E1 -25676.271,E2 -25676.271} C_VEL
LIN {X 0,Y 132.264,Z 299.284,A -85,B 0,C 180,E1 -25681.77,E2 -25681.77} C_VEL
LIN {X 0,Y 137.518,Z 294.555,A -85,B 0,C 180,E1 -25685.994,E2 -25685.994} C_VEL
LIN {X 0,Y 144.277,Z 287.812,A -85,B 0,C 180,E1 -25690.197,E2 -25690.197} C_VEL
LIN {X 0,Y 148.066,Z 283.622,A -85,B 0,C 180,E1 -25692.181,E2 -25692.181} C_VEL
LIN {X 0,Y 149.528,Z 281.366,A -85,B 0,C 180,E1 -25693.321,E2 -25693.321} C_VEL
LIN {X 0,Y 151.581,Z 273.935,A -85,B 0,C 180,E1 -25697.559,E2 -25697.559} C_VEL
LIN {X 0,Y 153.184,Z 271.302,A -85,B 0,C 180,E1 -25698.5,E2 -25698.5} C_VEL
LIN {X 0,Y 157.802,Z 264.643,A -85,B 0,C 180,E1 -25700.196,E2 -25700.196} C_VEL
LIN {X 0,Y 163.734,Z 255.021,A -85,B 0,C 180,E1 -25702.064,E2 -25702.064} C_VEL
LIN {X 0,Y 169.224,Z 244.517,A -85,B 0,C 180,E1 -25703.576,E2 -25703.576} C_VEL
LIN {X 0,Y 174.136,Z 232.905,A -85,B 0,C 180,E1 -25704.811,E2 -25704.811} C_VEL
LIN {X 0,Y 178.342,Z 219.628,A -85,B 0,C 180,E1 -25705.847,E2 -25705.847} C_VEL
LIN {X 0,Y 181.264,Z 206.425,A -85,B 0,C 180,E1 -25706.553,E2 -25706.553} C_VEL
LIN {X 0,Y 183.129,Z 190.936,A -85,B 0,C 180,E1 -25707.081,E2 -25707.081} C_VEL
LIN {X 0,Y 183.315,Z 188.082,A -85,B 0,C 180,E1 -25707.213,E2 -25707.213} C_VEL
LIN {X 0,Y 180.635,Z 180.286,A -85,B 0,C 180,E1 -25709.694,E2 -25709.694} C_VEL
LIN {X 0,Y 177.904,Z 173.114,A -85,B 0,C 180,E1 -25712.503,E2 -25712.503} C_VEL
LIN {X 0,Y 175.297,Z 166.896,A -85,B 0,C 180,E1 -25715.579,E2 -25715.579} C_VEL
LIN {X 0,Y 173.167,Z 162.091,A -85,B 0,C 180,E1 -25718.576,E2 -25718.576} C_VEL
LIN {X 0,Y 171.443,Z 158.192,A -85,B 0,C 180,E1 -25721.67,E2 -25721.67} C_VEL
LIN {X 0,Y 169.178,Z 153.196,A -85,B 0,C 180,E1 -25728.012,E2 -25728.012} C_VEL
LIN {X 0,Y 168.462,Z 152.697,A -85,B 0,C 180,E1 -25732.811,E2 -25732.811} C_VEL
LIN {X 0,Y 169.246,Z 153.012,A -85,B 0,C 180,E1 -25738.931,E2 -25738.931} C_VEL
LIN {X 0,Y 170.792,Z 156.55,A -85,B 0,C 180,E1 -25743.649,E2 -25743.649} C_VEL
LIN {X 0,Y 171.718,Z 157.858,A -85,B 0,C 180,E1 -25745.468,E2 -25745.468} C_VEL
LIN {X 0,Y 174.409,Z 162.591,A -85,B 0,C 180,E1 -25749.713,E2 -25749.713} C_VEL
LIN {X 0,Y 176.634,Z 166.482,A -85,B 0,C 180,E1 -25752.422,E2 -25752.422} C_VEL
LIN {X 0,Y 179.789,Z 172.154,A -85,B 0,C 180,E1 -25755.663,E2 -25755.663} C_VEL
LIN {X 0,Y 183.723,Z 180.042,A -85,B 0,C 180,E1 -25759.122,E2 -25759.122} C_VEL
LIN {X 0,Y 183.995,Z 181.072,A -85,B 0,C 180,E1 -25759.382,E2 -25759.382} C_VEL
LIN {X 0,Y 182.322,Z 196.062,A -85,B 0,C 180,E1 -25759.925,E2 -25759.925} C_VEL
LIN {X 0,Y 180.005,Z 207.82,A -85,B 0,C 180,E1 -25760.573,E2 -25760.573} C_VEL
LIN {X 0,Y 176.515,Z 220.409,A -85,B 0,C 180,E1 -25761.64,E2 -25761.64} C_VEL
LIN {X 0,Y 171.881,Z 232.816,A -85,B 0,C 180,E1 -25763.077,E2 -25763.077} C_VEL
LIN {X 0,Y 166.989,Z 243.223,A -85,B 0,C 180,E1 -25764.672,E2 -25764.672} C_VEL
LIN {X 0,Y 161.206,Z 253.256,A -85,B 0,C 180,E1 -25766.657,E2 -25766.657} C_VEL
LIN {X 0,Y 154.86,Z 262.551,A -85,B 0,C 180,E1 -25769.12,E2 -25769.12} C_VEL
LIN {X 0,Y 148.797,Z 270.157,A -85,B 0,C 180,E1 -25771.771,E2 -25771.771} C_VEL
LIN {X 0,Y 141.917,Z 277.562,A -85,B 0,C 180,E1 -25775.205,E2 -25775.205} C_VEL
LIN {X 0,Y 135.694,Z 283.395,A -85,B 0,C 180,E1 -25779.025,E2 -25779.025} C_VEL
LIN {X 0,Y 130.038,Z 287.917,A -85,B 0,C 180,E1 -25783.147,E2 -25783.147} C_VEL
LIN {X 0,Y 125.054,Z 291.284,A -85,B 0,C 180,E1 -25787.595,E2 -25787.595} C_VEL
LIN {X 0,Y 122.148,Z 292.926,A -85,B 0,C 180,E1 -25790.737,E2 -25790.737} C_VEL
LIN {X 0,Y 118.036,Z 294.733,A -85,B 0,C 180,E1 -25796.47,E2 -25796.47} C_VEL
LIN {X 0,Y 115.685,Z 295.234,A -85,B 0,C 180,E1 -25800.923,E2 -25800.923} C_VEL
LIN {X 0,Y 114.317,Z 295.157,A -85,B 0,C 180,E1 -25804.512,E2 -25804.512} C_VEL
LIN {X 0,Y 113.161,Z 294.56,A -85,B 0,C 180,E1 -25808.688,E2 -25808.688} C_VEL
LIN {X 0,Y 112.253,Z 292.41,A -85,B 0,C 180,E1 -25815.498,E2 -25815.498} C_VEL
LIN {X 0,Y 112.512,Z 289.585,A -85,B 0,C 180,E1 -25821.017,E2 -25821.017} C_VEL
LIN {X 0,Y 113.455,Z 285.731,A -85,B 0,C 180,E1 -25826.45,E2 -25826.45} C_VEL
LIN {X 0,Y 114.989,Z 280.758,A -85,B 0,C 180,E1 -25831.752,E2 -25831.752} C_VEL
LIN {X 0,Y 117.19,Z 274.519,A -85,B 0,C 180,E1 -25836.89,E2 -25836.89} C_VEL
LIN {X 0,Y 120.188,Z 266.736,A -85,B 0,C 180,E1 -25841.811,E2 -25841.811} C_VEL
LIN {X 0,Y 123.927,Z 256.974,A -85,B 0,C 180,E1 -25846.474,E2 -25846.474} C_VEL
LIN {X 0,Y 127.439,Z 247.194,A -85,B 0,C 180,E1 -25850.046,E2 -25850.046} C_VEL
LIN {X 0,Y 130.612,Z 236.904,A -85,B 0,C 180,E1 -25852.962,E2 -25852.962} C_VEL
LIN {X 0,Y 133.506,Z 226.067,A -85,B 0,C 180,E1 -25855.324,E2 -25855.324} C_VEL
LIN {X 0,Y 136.224,Z 214.086,A -85,B 0,C 180,E1 -25857.251,E2 -25857.251} C_VEL
LIN {X 0,Y 138.365,Z 201.071,A -85,B 0,C 180,E1 -25858.748,E2 -25858.748} C_VEL
LIN {X 0,Y 139.754,Z 187.599,A -85,B 0,C 180,E1 -25859.714,E2 -25859.714} C_VEL
LIN {X 0,Y 142.554,Z 144.681,A -85,B 0,C 180,E1 -25861.613,E2 -25861.613} C_VEL
LIN {X 0,Y 137.029,Z 132.71,A -85,B 0,C 180,E1 -25864.408,E2 -25864.408} C_VEL
LIN {X 0,Y 131.384,Z 122.511,A -85,B 0,C 180,E1 -25867.495,E2 -25867.495} C_VEL
LIN {X 0,Y 126.777,Z 115.423,A -85,B 0,C 180,E1 -25870.253,E2 -25870.253} C_VEL
LIN {X 0,Y 124.287,Z 111.773,A -85,B 0,C 180,E1 -25871.879,E2 -25871.879} C_VEL
LIN {X 0,Y 121.689,Z 108.147,A -85,B 0,C 180,E1 -25873.69,E2 -25873.69} C_VEL
LIN {X 0,Y 119.421,Z 105.361,A -85,B 0,C 180,E1 -25875.362,E2 -25875.362} C_VEL
LIN {X 0,Y 118.313,Z 103.451,A -85,B 0,C 180,E1 -25876.285,E2 -25876.285} C_VEL
LIN {X 0,Y 116.178,Z 101.512,A -85,B 0,C 180,E1 -25877.986,E2 -25877.986} C_VEL
LIN {X 0,Y 114.95,Z 98.915,A -85,B 0,C 180,E1 -25879.198,E2 -25879.198} C_VEL
LIN {X 0,Y 114.818,Z 98.168,A -85,B 0,C 180,E1 -25879.43,E2 -25879.43} C_VEL
LIN {X 0,Y 114.819,Z 98.124,A -85,B 0,C 180,E1 -25886.571,E2 -25886.571} C_VEL
LIN {X 0,Y 114.875,Z 98.173,A -85,B 0,C 180,E1 -25890.695,E2 -25890.695} C_VEL
LIN {X 0,Y 114.95,Z 98.148,A -85,B 0,C 180,E1 -25896.508,E2 -25896.508} C_VEL
LIN {X 0,Y 115.015,Z 98.143,A -85,B 0,C 180,E1 -25902.209,E2 -25902.209} C_VEL
LIN {X 0,Y 115.255,Z 98.127,A -85,B 0,C 180,E1 -25907.333,E2 -25907.333} C_VEL
LIN {X 0,Y 115.369,Z 98.096,A -85,B 0,C 180,E1 -25913.001,E2 -25913.001} C_VEL
LIN {X 0,Y 115.996,Z 98.016,A -85,B 0,C 180,E1 -25919.999,E2 -25919.999} C_VEL
LIN {X 0,Y 115.367,Z 98.099,A -85,B 0,C 180,E1 -25926.997,E2 -25926.997} C_VEL
LIN {X 0,Y 115.258,Z 98.127,A -85,B 0,C 180,E1 -25932.672,E2 -25932.672} C_VEL
LIN {X 0,Y 115.011,Z 98.153,A -85,B 0,C 180,E1 -25937.79,E2 -25937.79} C_VEL
LIN {X 0,Y 114.949,Z 98.166,A -85,B 0,C 180,E1 -25943.491,E2 -25943.491} C_VEL
LIN {X 0,Y 114.87,Z 98.17,A -85,B 0,C 180,E1 -25945.843,E2 -25945.843} C_VEL
LIN {X 0,Y 115.743,Z 100.801,A -85,B 0,C 180,E1 -25946.846,E2 -25946.846} C_VEL
LIN {X 0,Y 117.929,Z 103.166,A -85,B 0,C 180,E1 -25948.651,E2 -25948.651} C_VEL
LIN {X 0,Y 118.791,Z 103.946,A -85,B 0,C 180,E1 -25949.31,E2 -25949.31} C_VEL
LIN {X 0,Y 120.784,Z 107.15,A -85,B 0,C 180,E1 -25950.895,E2 -25950.895} C_VEL
